positionExtrema := output.trajectory.profiles[2].positionExtrema();
AssertEquals_LREAL(0.22338925049474447904, positionExtrema.Tmax, 1E-9, message:='Profile[2] Tmax incorrect');
AssertEquals_LREAL(94.47974487226861128875, positionExtrema.Maximum, 1E-9, message:='Profile[2] maximum incorrect');
AssertEquals_LREAL(0.02606362117094545780, positionExtrema.Tmin, 1E-9, message:='Profile[2] Tmin incorrect');
AssertEquals_LREAL(-104.28684661857214166503, positionExtrema.Minimum, 1E-9, message:='Profile[2] minimum incorrect');
   

TEST_FINISHED();
END_METHOD

METHOD Test_Trajectory_32
VAR_INST
  ruckig : Struckig.Ruckig(0.001);
  input : Struckig.InputParameter(3) := (
    Synchronization := SynchronizationType.TimeSync,        
    MaxVelocity := [ 2000.00000000000000000000, 2000.00000000000000000000, 2000.00000000000000000000 ],
    MaxAcceleration := [ 20000.00000000000000000000, 20000.00000000000000000000, 20000.00000000000000000000 ],
    MaxJerk := [ 800000.00000000000000000000, 800000.00000000000000000000, 800000.00000000000000000000 ],
    CurrentPosition := [ -71.32072487430589546875, 75.77874394332496876814, -31.17619673281745917848 ],
    CurrentVelocity := [ -39.37043543026334191381, -314.80982911633589083067, -743.63983854388607142027 ],
    CurrentAcceleration := [ 918.61171848468075040728, -8240.24070744882010330912, 376.40421615367449703626 ],
    TargetPosition := [ -38.32577323859909057546, 76.88839801585137934126, 77.24450399202348194194 ],
    TargetVelocity := [ 0.00000000000000000000, 0.00000000000000000000, 0.00000000000000000000 ],
    TargetAcceleration := [ 0.00000000000000000000, 0.00000000000000000000, 0.00000000000000000000 ]
  );
  output : Struckig.OutputParameter;
  positionExtrema : Struckig.PositionExtremaDesc;
END_VAR
TEST('Trajectory_32');

ruckig.update(input, output);

// Check total duration of profiles
AssertEquals_LREAL(Expected := 0.22561874467077386308, Actual := output.Trajectory.Duration, DELTA := 1E-8, Message := 'Duration incorrect');

// Check duration for each phase
positionExtrema := output.trajectory.profiles[0].positionExtrema();
AssertEquals_LREAL(0.22561874467077389084, positionExtrema.Tmax, 1E-9, message:='Profile[0] Tmax incorrect');
AssertEquals_LREAL(-38.32577323859909057546, positionExtrema.Maximum, 1E-9, message:='Profile[0] maximum incorrect');
AssertEquals_LREAL(0.00883895720172546244, positionExtrema.Tmin, 1E-9, message:='Profile[0] Tmin incorrect');
AssertEquals_LREAL(-71.54075918203305661791, positionExtrema.Minimum, 1E-9, message:='Profile[0] minimum incorrect');

positionExtrema := output.trajectory.profiles[1].positionExtrema();
AssertEquals_LREAL(0.22561874448389260261, positionExtrema.Tmax, 1E-9, message:='Profile[1] Tmax incorrect');
AssertEquals_LREAL(76.88839801585137934126, positionExtrema.Maximum, 1E-9, message:='Profile[1] maximum incorrect');
AssertEquals_LREAL(0.04326693976782886031, positionExtrema.Tmin, 1E-9, message:='Profile[1] Tmin incorrect');
AssertEquals_LREAL(64.99037106700389188063, positionExtrema.Minimum, 1E-9, message:='Profile[1] minimum incorrect');

positionExtrema := output.trajectory.profiles[2].positionExtrema();
AssertEquals_LREAL(0.22561874467077386308, positionExtrema.Tmax, 1E-9, message:='Profile[2] Tmax incorrect');
AssertEquals_LREAL(77.24450399202348194194, positionExtrema.Maximum, 1E-9, message:='Profile[2] maximum incorrect');
AssertEquals_LREAL(0.02452949472980790746, positionExtrema.Tmin, 1E-9, message:='Profile[2] Tmin incorrect');
AssertEquals_LREAL(-47.33615887649365561174, positionExtrema.Minimum, 1E-9, message:='Profile[2] minimum incorrect');
   

TEST_FINISHED();
END_METHOD

METHOD Test_Trajectory_33
VAR_INST
  ruckig : Struckig.Ruckig(0.001);
  input : Struckig.InputParameter(3) := (
    Synchronization := SynchronizationType.TimeSync,        
    MaxVelocity := [ 2000.00000000000000000000, 2000.00000000000000000000, 2000.00000000000000000000 ],
    MaxAcceleration := [ 20000.00000000000000000000, 20000.00000000000000000000, 20000.00000000000000000000 ],
    MaxJerk := [ 800000.00000000000000000000, 800000.00000000000000000000, 800000.00000000000000000000 ],
    CurrentPosition := [ -10.72081173000827902797, -58.44147038088563306246, 98.86324493851924444243 ],
    CurrentVelocity := [ -408.47451658779903027607, -786.19958599415508615493, -998.10812621012325962511 ],
    CurrentAcceleration := [ 3503.92425371204808470793, 3035.68280271572984929662, -8529.36175578239635797217 ],
    TargetPosition := [ -24.74505052699171869790, -29.66847304289291287205, -86.07591857423138037575 ],
    TargetVelocity := [ 0.00000000000000000000, 0.00000000000000000000, 0.00000000000000000000 ],
    TargetAcceleration := [ 0.00000000000000000000, 0.00000000000000000000, 0.00000000000000000000 ]
  );
  output : Struckig.OutputParameter;
  positionExtrema : Struckig.PositionExtremaDesc;
END_VAR
TEST('Trajectory_33');

ruckig.update(input, output);

// Check total duration of profiles
AssertEquals_LREAL(Expected := 0.17123630970102474147, Actual := output.Trajectory.Duration, DELTA := 1E-8, Message := 'Duration incorrect');

// Check duration for each phase
positionExtrema := output.trajectory.profiles[0].positionExtrema();
AssertEquals_LREAL(0.00000000000000000000, positionExtrema.Tmax, 1E-9, message:='Profile[0] Tmax incorrect');
AssertEquals_LREAL(-10.72081173000827902797, positionExtrema.Maximum, 1E-9, message:='Profile[0] maximum incorrect');
AssertEquals_LREAL(0.17123630970102476923, positionExtrema.Tmin, 1E-9, message:='Profile[0] Tmin incorrect');
AssertEquals_LREAL(-24.74505052699171869790, positionExtrema.Minimum, 1E-9, message:='Profile[0] minimum incorrect');

positionExtrema := output.trajectory.profiles[1].positionExtrema();
AssertEquals_LREAL(0.17123630970102471371, positionExtrema.Tmax, 1E-9, message:='Profile[1] Tmax incorrect');
AssertEquals_LREAL(-29.66847304289291287205, positionExtrema.Maximum, 1E-9, message:='Profile[1] maximum incorrect');
AssertEquals_LREAL(0.06908515615955748701, positionExtrema.Tmin, 1E-9, message:='Profile[1] Tmin incorrect');
AssertEquals_LREAL(-76.18339289032344652242, positionExtrema.Minimum, 1E-9, message:='Profile[1] minimum incorrect');

positionExtrema := output.trajectory.profiles[2].positionExtrema();
AssertEquals_LREAL(0.00000000000000000000, positionExtrema.Tmax, 1E-9, message:='Profile[2] Tmax incorrect');
AssertEquals_LREAL(98.86324493851924444243, positionExtrema.Maximum, 1E-9, message:='Profile[2] maximum incorrect');
AssertEquals_LREAL(0.17123630970102474147, positionExtrema.Tmin, 1E-9, message:='Profile[2] Tmin incorrect');
AssertEquals_LREAL(-86.07591857423138037575, positionExtrema.Minimum, 1E-9, message:='Profile[2] minimum incorrect');
   

TEST_FINISHED();
END_METHOD

METHOD Test_Trajectory_HasTargetVelocity_34
VAR_INST
  ruckig : Struckig.Ruckig(0.001);
  input : Struckig.InputParameter(3) := (
    Synchronization := SynchronizationType.TimeSync,        
    MaxVelocity := [ 2000.00000000000000000000, 2000.00000000000000000000, 2000.00000000000000000000 ],
    MaxAcceleration := [ 20000.00000000000000000000, 20000.00000000000000000000, 20000.00000000000000000000 ],
    MaxJerk := [ 800000.00000000000000000000, 800000.00000000000000000000, 800000.00000000000000000000 ],
    CurrentPosition := [ 52.72619781679460970736, -25.78201897219773286452, 80.53760009793651875043 ],
    CurrentVelocity := [ -120.69783207836667315860, 178.50171370384009605914, -265.96277737557261389156 ],
    CurrentAcceleration := [ 9869.62339068779328954406, 8236.73224664633380598389, 4587.35631399299018085003 ],
    TargetPosition := [ -7.31302355801524583967, 98.53124939615054245223, -70.22704739896117587250 ],
    TargetVelocity := [ 648.92680228108224582684, 640.55767309494626715605, -28.66025813343185291160 ],
    TargetAcceleration := [ 0.00000000000000000000, 0.00000000000000000000, 0.00000000000000000000 ]
  );
  output : Struckig.OutputParameter;
  positionExtrema : Struckig.PositionExtremaDesc;
END_VAR
TEST('Trajectory_HasTargetVelocity_34');

ruckig.update(input, output);

// Check total duration of profiles
AssertEquals_LREAL(Expected := 0.19340758597333415625, Actual := output.Trajectory.Duration, DELTA := 1E-8, Message := 'Duration incorrect');

// Check duration for each phase
positionExtrema := output.trajectory.profiles[0].positionExtrema();
AssertEquals_LREAL(0.00000000000000000000, positionExtrema.Tmax, 1E-9, message:='Profile[0] Tmax incorrect');
AssertEquals_LREAL(52.72619781679460970736, positionExtrema.Maximum, 1E-9, message:='Profile[0] maximum incorrect');
AssertEquals_LREAL(0.16840758597333416180, positionExtrema.Tmin, 1E-9, message:='Profile[0] Tmin incorrect');
AssertEquals_LREAL(-21.45286028170894354616, positionExtrema.Minimum, 1E-9, message:='Profile[0] minimum incorrect');

positionExtrema := output.trajectory.profiles[1].positionExtrema();
AssertEquals_LREAL(0.19340758597333415625, positionExtrema.Tmax, 1E-9, message:='Profile[1] Tmax incorrect');
AssertEquals_LREAL(98.53124939615054245223, positionExtrema.Maximum, 1E-9, message:='Profile[1] maximum incorrect');
AssertEquals_LREAL(0.00000000000000000000, positionExtrema.Tmin, 1E-9, message:='Profile[1] Tmin incorrect');
AssertEquals_LREAL(-25.78201897219773286452, positionExtrema.Minimum, 1E-9, message:='Profile[1] minimum incorrect');

positionExtrema := output.trajectory.profiles[2].positionExtrema();
AssertEquals_LREAL(0.00000000000000000000, positionExtrema.Tmax, 1E-9, message:='Profile[2] Tmax incorrect');
AssertEquals_LREAL(80.53760009793651875043, positionExtrema.Maximum, 1E-9, message:='Profile[2] maximum incorrect');
AssertEquals_LREAL(0.19340758597333415625, positionExtrema.Tmin, 1E-9, message:='Profile[2] Tmin incorrect');
AssertEquals_LREAL(-70.22704739896117587250, positionExtrema.Minimum, 1E-9, message:='Profile[2] minimum incorrect');
   

TEST_FINISHED();
END_METHOD

METHOD Test_Trajectory_HasTargetVelocity_35
VAR_INST
  ruckig : Struckig.Ruckig(0.001);
  input : Struckig.InputParameter(3) := (
    Synchronization := SynchronizationType.TimeSync,        
    MaxVelocity := [ 2000.00000000000000000000, 2000.00000000000000000000, 2000.00000000000000000000 ],
    MaxAcceleration := [ 20000.00000000000000000000, 20000.00000000000000000000, 20000.00000000000000000000 ],
    MaxJerk := [ 800000.00000000000000000000, 800000.00000000000000000000, 800000.00000000000000000000 ],
    CurrentPosition := [ -34.17551015513085133080, -36.11913195800440234962, 51.20006403327516864010 ],
    CurrentVelocity := [ -436.11356880285654824547, -175.40667275745920505869, 746.11367552095180144534 ],
    CurrentAcceleration := [ -9866.78282408208724518772, -2137.40956356850620068144, 2870.77810427219810662791 ],
    TargetPosition := [ 94.89098874895094581916, -43.87608688101931875281, 99.33475834942979076914 ],
    TargetVelocity := [ 945.80038372223793885496, -169.18944510068342879094, 349.24092684862353053177 ],
    TargetAcceleration := [ 0.00000000000000000000, 0.00000000000000000000, 0.00000000000000000000 ]
  );
  output : Struckig.OutputParameter;
  positionExtrema : Struckig.PositionExtremaDesc;
END_VAR
TEST('Trajectory_HasTargetVelocity_35');

ruckig.update(input, output);

// Check total duration of profiles
AssertEquals_LREAL(Expected := 0.19433376507479860340, Actual := output.Trajectory.Duration, DELTA := 1E-8, Message := 'Duration incorrect');

// Check duration for each phase
positionExtrema := output.trajectory.profiles[0].positionExtrema();
AssertEquals_LREAL(0.19433376507479860340, positionExtrema.Tmax, 1E-9, message:='Profile[0] Tmax incorrect');
AssertEquals_LREAL(94.89098874895094581916, positionExtrema.Maximum, 1E-9, message:='Profile[0] maximum incorrect');
AssertEquals_LREAL(0.03733347853010261091, positionExtrema.Tmin, 1E-9, message:='Profile[0] Tmin incorrect');
AssertEquals_LREAL(-50.39525451816182055609, positionExtrema.Minimum, 1E-9, message:='Profile[0] minimum incorrect');

positionExtrema := output.trajectory.profiles[1].positionExtrema();
AssertEquals_LREAL(0.00000000000000000000, positionExtrema.Tmax, 1E-9, message:='Profile[1] Tmax incorrect');
AssertEquals_LREAL(-36.11913195800440234962, positionExtrema.Maximum, 1E-9, message:='Profile[1] maximum incorrect');
AssertEquals_LREAL(0.19433376507479860340, positionExtrema.Tmin, 1E-9, message:='Profile[1] Tmin incorrect');
AssertEquals_LREAL(-43.87608688101931875281, positionExtrema.Minimum, 1E-9, message:='Profile[1] minimum incorrect');

positionExtrema := output.trajectory.profiles[2].positionExtrema();
AssertEquals_LREAL(0.19433376507479860340, positionExtrema.Tmax, 1E-9, message:='Profile[2] Tmax incorrect');
AssertEquals_LREAL(99.33475834942979076914, positionExtrema.Maximum, 1E-9, message:='Profile[2] maximum incorrect');
AssertEquals_LREAL(0.00000000000000000000, positionExtrema.Tmin, 1E-9, message:='Profile[2] Tmin incorrect');
AssertEquals_LREAL(51.20006403327516864010, positionExtrema.Minimum, 1E-9, message:='Profile[2] minimum incorrect');
   

TEST_FINISHED();
END_METHOD

METHOD Test_Trajectory_HasTargetVelocity_36
VAR_INST
  ruckig : Struckig.Ruckig(0.001);
  input : Struckig.InputParameter(3) := (
    Synchronization := SynchronizationType.TimeSync,        
    MaxVelocity := [ 2000.00000000000000000000, 2000.00000000000000000000, 2000.00000000000000000000 ],
    MaxAcceleration := [ 20000.00000000000000000000, 20000.00000000000000000000, 20000.00000000000000000000 ],
    MaxJerk := [ 800000.00000000000000000000, 800000.00000000000000000000, 800000.00000000000000000000 ],
    CurrentPosition := [ 64.35804589046725254775, -17.92542582379405757820, 1.48297994216896711350 ],
    CurrentVelocity := [ 464.92943892208950273925, -779.25597761349285974575, 998.42982599227457285451 ],
    CurrentAcceleration := [ 4749.41918638301285682246, -6355.94416374630964128301, 521.38908747176901670173 ],
    TargetPosition := [ 90.33897695077399703223, -51.53109090258827507114, -18.12118447758692241223 ],
    TargetVelocity := [ 651.93427968717173826008, 22.75188801650608638738, 576.72189974234174769663 ],
    TargetAcceleration := [ 0.00000000000000000000, 0.00000000000000000000, 0.00000000000000000000 ]
  );
  output : Struckig.OutputParameter;
  positionExtrema : Struckig.PositionExtremaDesc;
END_VAR
TEST('Trajectory_HasTargetVelocity_36');

ruckig.update(input, output);

// Check total duration of profiles
AssertEquals_LREAL(Expected := 0.22796271730102146691, Actual := output.Trajectory.Duration, DELTA := 1E-8, Message := 'Duration incorrect');

// Check duration for each phase
positionExtrema := output.trajectory.profiles[0].positionExtrema();
AssertEquals_LREAL(0.22796271730102146691, positionExtrema.Tmax, 1E-9, message:='Profile[0] Tmax incorrect');
AssertEquals_LREAL(90.33897695077399703223, positionExtrema.Maximum, 1E-9, message:='Profile[0] maximum incorrect');
AssertEquals_LREAL(0.00000000000000000000, positionExtrema.Tmin, 1E-9, message:='Profile[0] Tmin incorrect');
AssertEquals_LREAL(64.35804589046725254775, positionExtrema.Minimum, 1E-9, message:='Profile[0] minimum incorrect');

positionExtrema := output.trajectory.profiles[1].positionExtrema();
AssertEquals_LREAL(0.00000000000000000000, positionExtrema.Tmax, 1E-9, message:='Profile[1] Tmax incorrect');
AssertEquals_LREAL(-17.92542582379405757820, positionExtrema.Maximum, 1E-9, message:='Profile[1] maximum incorrect');
AssertEquals_LREAL(0.21997970156554483290, positionExtrema.Tmin, 1E-9, message:='Profile[1] Tmin incorrect');
AssertEquals_LREAL(-51.64657663770686468752, positionExtrema.Minimum, 1E-9, message:='Profile[1] minimum incorrect');

positionExtrema := output.trajectory.profiles[2].positionExtrema();
AssertEquals_LREAL(0.09985417258924977890, positionExtrema.Tmax, 1E-9, message:='Profile[2] Tmax incorrect');
AssertEquals_LREAL(25.50333501341721742506, positionExtrema.Maximum, 1E-9, message:='Profile[2] maximum incorrect');
AssertEquals_LREAL(0.20296271730102147246, positionExtrema.Tmin, 1E-9, message:='Profile[2] Tmin incorrect');
AssertEquals_LREAL(-30.45589863781214745586, positionExtrema.Minimum, 1E-9, message:='Profile[2] minimum incorrect');
   

TEST_FINISHED();
END_METHOD

METHOD Test_Trajectory_HasTargetAcceleration_37
VAR_INST
  ruckig : Struckig.Ruckig(0.001);
  input : Struckig.InputParameter(3) := (
    Synchronization := SynchronizationType.TimeSync,        
    MaxVelocity := [ 2000.00000000000000000000, 2000.00000000000000000000, 2000.00000000000000000000 ],
    MaxAcceleration := [ 20000.00000000000000000000, 20000.00000000000000000000, 20000.00000000000000000000 ],
    MaxJerk := [ 800000.00000000000000000000, 800000.00000000000000000000, 800000.00000000000000000000 ],
    CurrentPosition := [ 75.70258410717627839404, -31.81448222562724481577, -58.08554852109006816363 ],
    CurrentVelocity := [ 171.95882136884461033333, -584.70058950900761374214, 745.12321825604590230796 ],
    CurrentAcceleration := [ 5092.19654988173533638474, 7179.19572851603152230382, 1704.28450887377948674839 ],
    TargetPosition := [ 97.60417669221266123714, 88.97844242319803242935, -19.79432812800784802221 ],
    TargetVelocity := [ 0.00000000000000000000, 0.00000000000000000000, 0.00000000000000000000 ],
    TargetAcceleration := [ 983.95730849860865419032, -389.38723727042054179037, -311.43162034307158592128 ]
  );
  output : Struckig.OutputParameter;
  positionExtrema : Struckig.PositionExtremaDesc;
END_VAR
TEST('Trajectory_HasTargetAcceleration_37');

ruckig.update(input, output);

// Check total duration of profiles
AssertEquals_LREAL(Expected := 0.21113509394885510151, Actual := output.Trajectory.Duration, DELTA := 1E-8, Message := 'Duration incorrect');

// Check duration for each phase
positionExtrema := output.trajectory.profiles[0].positionExtrema();
AssertEquals_LREAL(0.20867520067760855773, positionExtrema.Tmax, 1E-9, message:='Profile[0] Tmax incorrect');
AssertEquals_LREAL(97.60516902544232209493, positionExtrema.Maximum, 1E-9, message:='Profile[0] maximum incorrect');
AssertEquals_LREAL(0.00000000000000000000, positionExtrema.Tmin, 1E-9, message:='Profile[0] Tmin incorrect');
AssertEquals_LREAL(75.70258410717627839404, positionExtrema.Minimum, 1E-9, message:='Profile[0] minimum incorrect');

positionExtrema := output.trajectory.profiles[1].positionExtrema();
AssertEquals_LREAL(0.21113509394885510151, positionExtrema.Tmax, 1E-9, message:='Profile[1] Tmax incorrect');
AssertEquals_LREAL(88.97844242319803242935, positionExtrema.Maximum, 1E-9, message:='Profile[1] maximum incorrect');
AssertEquals_LREAL(0.01602600533935496022, positionExtrema.Tmin, 1E-9, message:='Profile[1] Tmin incorrect');
AssertEquals_LREAL(-39.71416974486287898571, positionExtrema.Minimum, 1E-9, message:='Profile[1] minimum incorrect');

positionExtrema := output.trajectory.profiles[2].positionExtrema();
AssertEquals_LREAL(0.21113509394885504600, positionExtrema.Tmax, 1E-9, message:='Profile[2] Tmax incorrect');
AssertEquals_LREAL(-19.79432812800784091678, positionExtrema.Maximum, 1E-9, message:='Profile[2] maximum incorrect');
AssertEquals_LREAL(0.00000000000000000000, positionExtrema.Tmin, 1E-9, message:='Profile[2] Tmin incorrect');
AssertEquals_LREAL(-58.08554852109006816363, positionExtrema.Minimum, 1E-9, message:='Profile[2] minimum incorrect');
   

TEST_FINISHED();
END_METHOD

METHOD Test_Trajectory_HasTargetVelocity_HasTargetAcceleration_38
VAR_INST
  ruckig : Struckig.Ruckig(0.001);
  input : Struckig.InputParameter(3) := (
    Synchronization := SynchronizationType.TimeSync,        
    MaxVelocity := [ 2000.00000000000000000000, 2000.00000000000000000000, 2000.00000000000000000000 ],
    MaxAcceleration := [ 20000.00000000000000000000, 20000.00000000000000000000, 20000.00000000000000000000 ],
    MaxJerk := [ 800000.00000000000000000000, 800000.00000000000000000000, 800000.00000000000000000000 ],
    CurrentPosition := [ 70.18836201933098095651, -77.67370458831963730972, -11.76145133517785268396 ],
    CurrentVelocity := [ -105.04558581308560860634, 265.56449346599174532457, 964.37814674831179218017 ],
    CurrentAcceleration := [ -6039.95733145092708582524, -2777.20507650207400729414, 4352.81085492715828877408 ],
    TargetPosition := [ 71.40233970199534496714, 5.40303445887771260914, 92.98580498819549688960 ],
    TargetVelocity := [ -236.50355991826609169948, -66.98837676043160627160, 870.41763001953563616553 ],
    TargetAcceleration := [ -500.07275325607560034769, 72.93763981243137095589, -942.49209154303241575690 ]
  );
  output : Struckig.OutputParameter;
  positionExtrema : Struckig.PositionExtremaDesc;
END_VAR
TEST('Trajectory_HasTargetVelocity_HasTargetAcceleration_38');

ruckig.update(input, output);

// Check total duration of profiles
AssertEquals_LREAL(Expected := 0.14901888909886754075, Actual := output.Trajectory.Duration, DELTA := 1E-8, Message := 'Duration incorrect');

// Check duration for each phase
positionExtrema := output.trajectory.profiles[0].positionExtrema();
AssertEquals_LREAL(0.12406814159805865105, positionExtrema.Tmax, 1E-9, message:='Profile[0] Tmax incorrect');
AssertEquals_LREAL(75.12313380408009777511, positionExtrema.Maximum, 1E-9, message:='Profile[0] maximum incorrect');
AssertEquals_LREAL(0.02561480747291104351, positionExtrema.Tmin, 1E-9, message:='Profile[0] Tmin incorrect');
AssertEquals_LREAL(67.75537848504214366585, positionExtrema.Minimum, 1E-9, message:='Profile[0] minimum incorrect');

positionExtrema := output.trajectory.profiles[1].positionExtrema();
AssertEquals_LREAL(0.13598633944686283614, positionExtrema.Tmax, 1E-9, message:='Profile[1] Tmax incorrect');
AssertEquals_LREAL(5.98711873384755755012, positionExtrema.Maximum, 1E-9, message:='Profile[1] maximum incorrect');
AssertEquals_LREAL(0.00000000000000000000, positionExtrema.Tmin, 1E-9, message:='Profile[1] Tmin incorrect');
AssertEquals_LREAL(-77.67370458831963730972, positionExtrema.Minimum, 1E-9, message:='Profile[1] minimum incorrect');

positionExtrema := output.trajectory.profiles[2].positionExtrema();
AssertEquals_LREAL(0.14901888909886754075, positionExtrema.Tmax, 1E-9, message:='Profile[2] Tmax incorrect');
AssertEquals_LREAL(92.98580498819549688960, positionExtrema.Maximum, 1E-9, message:='Profile[2] maximum incorrect');
AssertEquals_LREAL(0.00000000000000000000, positionExtrema.Tmin, 1E-9, message:='Profile[2] Tmin incorrect');
AssertEquals_LREAL(-11.76145133517785268396, positionExtrema.Minimum, 1E-9, message:='Profile[2] minimum incorrect');
   

TEST_FINISHED();
END_METHOD

METHOD Test_Trajectory_HasTargetAcceleration_39
VAR_INST
  ruckig : Struckig.Ruckig(0.001);
  input : Struckig.InputParameter(3) := (
    Synchronization := SynchronizationType.TimeSync,        
    MaxVelocity := [ 2000.00000000000000000000, 2000.00000000000000000000, 2000.00000000000000000000 ],
    MaxAcceleration := [ 20000.00000000000000000000, 20000.00000000000000000000, 20000.00000000000000000000 ],
    MaxJerk := [ 800000.00000000000000000000, 800000.00000000000000000000, 800000.00000000000000000000 ],
    CurrentPosition := [ -21.93974605417949419461, -18.49856402298217972202, -96.65992156980888694306 ],
    CurrentVelocity := [ 560.92968123589912465832, -454.79210991651348194864, -556.36905002756998328550 ],
    CurrentAcceleration := [ 6747.73447463338743546046, 9628.82123479624351602979, 5462.73061834566397010349 ],
    TargetPosition := [ -36.27372063241573840742, 69.45477693939508867516, -56.03831440156044152445 ],
    TargetVelocity := [ 0.00000000000000000000, 0.00000000000000000000, 0.00000000000000000000 ],
    TargetAcceleration := [ 228.31394350642813151353, -518.68886336123591718206, -694.01647177787629061640 ]
  );
  output : Struckig.OutputParameter;
  positionExtrema : Struckig.PositionExtremaDesc;
END_VAR
TEST('Trajectory_HasTargetAcceleration_39');

ruckig.update(input, output);

// Check total duration of profiles
AssertEquals_LREAL(Expected := 0.17804896497402217248, Actual := output.Trajectory.Duration, DELTA := 1E-8, Message := 'Duration incorrect');

// Check duration for each phase
positionExtrema := output.trajectory.profiles[0].positionExtrema();
AssertEquals_LREAL(0.05596801189631349371, positionExtrema.Tmax, 1E-9, message:='Profile[0] Tmax incorrect');
AssertEquals_LREAL(-1.82711489240683677693, positionExtrema.Maximum, 1E-9, message:='Profile[0] maximum incorrect');
AssertEquals_LREAL(0.17804896497402203370, positionExtrema.Tmin, 1E-9, message:='Profile[0] Tmin incorrect');
AssertEquals_LREAL(-36.27372063241574551284, positionExtrema.Minimum, 1E-9, message:='Profile[0] minimum incorrect');

positionExtrema := output.trajectory.profiles[1].positionExtrema();
AssertEquals_LREAL(0.17804896497402217248, positionExtrema.Tmax, 1E-9, message:='Profile[1] Tmax incorrect');
AssertEquals_LREAL(69.45477693939508867516, positionExtrema.Maximum, 1E-9, message:='Profile[1] maximum incorrect');
AssertEquals_LREAL(0.01296397345650469532, positionExtrema.Tmin, 1E-9, message:='Profile[1] Tmin incorrect');
AssertEquals_LREAL(-23.29484015015810172144, positionExtrema.Minimum, 1E-9, message:='Profile[1] minimum incorrect');

positionExtrema := output.trajectory.profiles[2].positionExtrema();
AssertEquals_LREAL(0.17804896497402220024, positionExtrema.Tmax, 1E-9, message:='Profile[2] Tmax incorrect');
AssertEquals_LREAL(-56.03831440156044152445, positionExtrema.Maximum, 1E-9, message:='Profile[2] maximum incorrect');
AssertEquals_LREAL(0.04613976266622405592, positionExtrema.Tmin, 1E-9, message:='Profile[2] Tmin incorrect');
AssertEquals_LREAL(-106.33609120894020350079, positionExtrema.Minimum, 1E-9, message:='Profile[2] minimum incorrect');
   

TEST_FINISHED();
END_METHOD

METHOD Test_Trajectory_40
VAR_INST
  ruckig : Struckig.Ruckig(0.001);
  input : Struckig.InputParameter(3) := (
    Synchronization := SynchronizationType.TimeSync,        
    MaxVelocity := [ 2000.00000000000000000000, 2000.00000000000000000000, 2000.00000000000000000000 ],
    MaxAcceleration := [ 20000.00000000000000000000, 20000.00000000000000000000, 20000.00000000000000000000 ],
    MaxJerk := [ 800000.00000000000000000000, 800000.00000000000000000000, 800000.00000000000000000000 ],
    CurrentPosition := [ 29.38520952151498022431, 0.54024576846694571941, -55.20826603737940274641 ],
    CurrentVelocity := [ -969.77050425776712927473, -274.95655325444397476531, 136.62875181670483470953 ],
    CurrentAcceleration := [ -3024.14261213553436391521, 816.78995976388432609383, -4328.68204209528175852029 ],
    TargetPosition := [ 1.97730433317153142525, -41.44239712071811254646, -63.08579022434781791162 ],
    TargetVelocity := [ 0.00000000000000000000, 0.00000000000000000000, 0.00000000000000000000 ],
    TargetAcceleration := [ 0.00000000000000000000, 0.00000000000000000000, 0.00000000000000000000 ]
  );
  output : Struckig.OutputParameter;
  positionExtrema : Struckig.PositionExtremaDesc;
END_VAR
TEST('Trajectory_40');

ruckig.update(input, output);

// Check total duration of profiles
AssertEquals_LREAL(Expected := 0.13217815288228063064, Actual := output.Trajectory.Duration, DELTA := 1E-8, Message := 'Duration incorrect');

// Check duration for each phase
positionExtrema := output.trajectory.profiles[0].positionExtrema();
AssertEquals_LREAL(0.00000000000000000000, positionExtrema.Tmax, 1E-9, message:='Profile[0] Tmax incorrect');
AssertEquals_LREAL(29.38520952151498022431, positionExtrema.Maximum, 1E-9, message:='Profile[0] maximum incorrect');
AssertEquals_LREAL(0.06794606535212494025, positionExtrema.Tmin, 1E-9, message:='Profile[0] Tmin incorrect');
AssertEquals_LREAL(-9.67357879957821609196, positionExtrema.Minimum, 1E-9, message:='Profile[0] minimum incorrect');

positionExtrema := output.trajectory.profiles[1].positionExtrema();
AssertEquals_LREAL(0.00000000000000000000, positionExtrema.Tmax, 1E-9, message:='Profile[1] Tmax incorrect');
AssertEquals_LREAL(0.54024576846694571941, positionExtrema.Maximum, 1E-9, message:='Profile[1] maximum incorrect');
AssertEquals_LREAL(0.13217815288228063064, positionExtrema.Tmin, 1E-9, message:='Profile[1] Tmin incorrect');
AssertEquals_LREAL(-41.44239712071811254646, positionExtrema.Minimum, 1E-9, message:='Profile[1] minimum incorrect');

positionExtrema := output.trajectory.profiles[2].positionExtrema();
AssertEquals_LREAL(0.01413581147570610458, positionExtrema.Tmax, 1E-9, message:='Profile[2] Tmax incorrect');
AssertEquals_LREAL(-54.08246211603182018735, positionExtrema.Maximum, 1E-9, message:='Profile[2] maximum incorrect');
AssertEquals_LREAL(0.13217815261799065185, positionExtrema.Tmin, 1E-9, message:='Profile[2] Tmin incorrect');
AssertEquals_LREAL(-63.08579022434781791162, positionExtrema.Minimum, 1E-9, message:='Profile[2] minimum incorrect');
   

TEST_FINISHED();
END_METHOD

METHOD Test_Trajectory_HasTargetVelocity_HasTargetAcceleration_41
VAR_INST
  ruckig : Struckig.Ruckig(0.001);
  input : Struckig.InputParameter(3) := (
    Synchronization := SynchronizationType.TimeSync,        
    MaxVelocity := [ 2000.00000000000000000000, 2000.00000000000000000000, 2000.00000000000000000000 ],
    MaxAcceleration := [ 20000.00000000000000000000, 20000.00000000000000000000, 20000.00000000000000000000 ],
    MaxJerk := [ 800000.00000000000000000000, 800000.00000000000000000000, 800000.00000000000000000000 ],
    CurrentPosition := [ 77.70133891525995295524, 7.01592092562633240505, 41.88398938907070601090 ],
    CurrentVelocity := [ -954.47536643469038608600, -572.16261829852851406031, 473.16402135503631143365 ],
    CurrentAcceleration := [ -2847.17654342300011194311, -1889.61698757276462856680, -3110.21768918452016805531 ],
    TargetPosition := [ 92.37579717709354554245, -14.04614057772144519731, -73.88361356505039623244 ],
    TargetVelocity := [ 519.95772801058456025203, 127.89327712966064609645, -380.91422286825297760515 ],
    TargetAcceleration := [ -890.64075852453197512659, 681.51569675393488978443, 390.99828361762297390669 ]
  );
  output : Struckig.OutputParameter;
  positionExtrema : Struckig.PositionExtremaDesc;
END_VAR
TEST('Trajectory_HasTargetVelocity_HasTargetAcceleration_41');

ruckig.update(input, output);

// Check total duration of profiles
AssertEquals_LREAL(Expected := 0.18543052523247699481, Actual := output.Trajectory.Duration, DELTA := 1E-8, Message := 'Duration incorrect');

// Check duration for each phase
positionExtrema := output.trajectory.profiles[0].positionExtrema();
AssertEquals_LREAL(0.18543052523247699481, positionExtrema.Tmax, 1E-9, message:='Profile[0] Tmax incorrect');
AssertEquals_LREAL(92.37579717709354554245, positionExtrema.Maximum, 1E-9, message:='Profile[0] maximum incorrect');
AssertEquals_LREAL(0.07568410654937982041, positionExtrema.Tmin, 1E-9, message:='Profile[0] Tmin incorrect');
AssertEquals_LREAL(41.15768150995504015555, positionExtrema.Minimum, 1E-9, message:='Profile[0] minimum incorrect');

positionExtrema := output.trajectory.profiles[1].positionExtrema();
AssertEquals_LREAL(0.00000000000000000000, positionExtrema.Tmax, 1E-9, message:='Profile[1] Tmax incorrect');
AssertEquals_LREAL(7.01592092562633240505, positionExtrema.Maximum, 1E-9, message:='Profile[1] maximum incorrect');
AssertEquals_LREAL(0.16752625845292970497, positionExtrema.Tmin, 1E-9, message:='Profile[1] Tmin incorrect');
AssertEquals_LREAL(-15.47801998831725711625, positionExtrema.Minimum, 1E-9, message:='Profile[1] minimum incorrect');

positionExtrema := output.trajectory.profiles[2].positionExtrema();
AssertEquals_LREAL(0.02111222788851935261, positionExtrema.Tmax, 1E-9, message:='Profile[2] Tmax incorrect');
AssertEquals_LREAL(49.92568034606993876423, positionExtrema.Maximum, 1E-9, message:='Profile[2] maximum incorrect');
AssertEquals_LREAL(0.18543052523247699481, positionExtrema.Tmin, 1E-9, message:='Profile[2] Tmin incorrect');
AssertEquals_LREAL(-73.88361356505039623244, positionExtrema.Minimum, 1E-9, message:='Profile[2] minimum incorrect');
   

TEST_FINISHED();
END_METHOD

METHOD Test_Trajectory_HasTargetAcceleration_42
VAR_INST
  ruckig : Struckig.Ruckig(0.001);
  input : Struckig.InputParameter(3) := (
    Synchronization := SynchronizationType.TimeSync,        
    MaxVelocity := [ 2000.00000000000000000000, 2000.00000000000000000000, 2000.00000000000000000000 ],
    MaxAcceleration := [ 20000.00000000000000000000, 20000.00000000000000000000, 20000.00000000000000000000 ],
    MaxJerk := [ 800000.00000000000000000000, 800000.00000000000000000000, 800000.00000000000000000000 ],
    CurrentPosition := [ 1.58314797372935345265, 90.58707779544036498010, 7.41484167737418431443 ],
    CurrentVelocity := [ 264.66369378964441239077, -967.86838256043972705811, 875.55912471800957064261 ],
    CurrentAcceleration := [ -5955.60883189429478079546, -8419.85921682317348313518, 8392.40723541911211214028 ],
    TargetPosition := [ -58.56616862494692554719, 73.15314018228875170280, 71.09694589628986705065 ],
    TargetVelocity := [ 0.00000000000000000000, 0.00000000000000000000, 0.00000000000000000000 ],
    TargetAcceleration := [ -714.77249466642297193175, -738.86959085233320365660, -949.40990195438507726067 ]
  );
  output : Struckig.OutputParameter;
  positionExtrema : Struckig.PositionExtremaDesc;
END_VAR
TEST('Trajectory_HasTargetAcceleration_42');

ruckig.update(input, output);

// Check total duration of profiles
AssertEquals_LREAL(Expected := 0.16824213942746521488, Actual := output.Trajectory.Duration, DELTA := 1E-8, Message := 'Duration incorrect');

// Check duration for each phase
positionExtrema := output.trajectory.profiles[0].positionExtrema();
AssertEquals_LREAL(0.01755548896013213109, positionExtrema.Tmax, 1E-9, message:='Profile[0] Tmax incorrect');
AssertEquals_LREAL(4.59030121571332649921, positionExtrema.Maximum, 1E-9, message:='Profile[0] maximum incorrect');
AssertEquals_LREAL(0.16645520819079967501, positionExtrema.Tmin, 1E-9, message:='Profile[0] Tmin incorrect');
AssertEquals_LREAL(-58.56654901772477472832, positionExtrema.Minimum, 1E-9, message:='Profile[0] minimum incorrect');

positionExtrema := output.trajectory.profiles[1].positionExtrema();
AssertEquals_LREAL(0.00000000000000000000, positionExtrema.Tmax, 1E-9, message:='Profile[1] Tmax incorrect');
AssertEquals_LREAL(90.58707779544036498010, positionExtrema.Maximum, 1E-9, message:='Profile[1] maximum incorrect');
AssertEquals_LREAL(0.09014117386002259980, positionExtrema.Tmin, 1E-9, message:='Profile[1] Tmin incorrect');
AssertEquals_LREAL(45.07056608531748764790, positionExtrema.Minimum, 1E-9, message:='Profile[1] minimum incorrect');

positionExtrema := output.trajectory.profiles[2].positionExtrema();
AssertEquals_LREAL(0.13468422806677898818, positionExtrema.Tmax, 1E-9, message:='Profile[2] Tmax incorrect');
AssertEquals_LREAL(73.02284673044322005353, positionExtrema.Maximum, 1E-9, message:='Profile[2] maximum incorrect');
AssertEquals_LREAL(0.00000000000000000000, positionExtrema.Tmin, 1E-9, message:='Profile[2] Tmin incorrect');
AssertEquals_LREAL(7.41484167737418431443, positionExtrema.Minimum, 1E-9, message:='Profile[2] minimum incorrect');
   

TEST_FINISHED();
END_METHOD

METHOD Test_Trajectory_HasTargetAcceleration_43
VAR_INST
  ruckig : Struckig.Ruckig(0.001);
  input : Struckig.InputParameter(3) := (
    Synchronization := SynchronizationType.TimeSync,        
    MaxVelocity := [ 2000.00000000000000000000, 2000.00000000000000000000, 2000.00000000000000000000 ],
    MaxAcceleration := [ 20000.00000000000000000000, 20000.00000000000000000000, 20000.00000000000000000000 ],
    MaxJerk := [ 800000.00000000000000000000, 800000.00000000000000000000, 800000.00000000000000000000 ],
    CurrentPosition := [ 53.13739682938987130001, -22.44298053732963182938, -41.20042774153274223181 ],
    CurrentVelocity := [ -304.98663512538098530058, 35.02037430652057992120, 738.80078152761325327447 ],
    CurrentAcceleration := [ -7270.26712820171451312490, -845.41004591047749272548, -4566.56327336276262940373 ],
    TargetPosition := [ 81.86956314333414752582, 96.25424125499196748024, -65.78248687323761600965 ],
    TargetVelocity := [ 0.00000000000000000000, 0.00000000000000000000, 0.00000000000000000000 ],
    TargetAcceleration := [ -511.94239891635919548207, 447.91143210314089628810, -814.86235086373915237345 ]
  );
  output : Struckig.OutputParameter;
  positionExtrema : Struckig.PositionExtremaDesc;
END_VAR
TEST('Trajectory_HasTargetAcceleration_43');

ruckig.update(input, output);

// Check total duration of profiles
AssertEquals_LREAL(Expected := 0.18070492746146707419, Actual := output.Trajectory.Duration, DELTA := 1E-8, Message := 'Duration incorrect');

// Check duration for each phase
positionExtrema := output.trajectory.profiles[0].positionExtrema();
AssertEquals_LREAL(0.18070492746146707419, positionExtrema.Tmax, 1E-9, message:='Profile[0] Tmax incorrect');
AssertEquals_LREAL(81.86956314333414752582, positionExtrema.Maximum, 1E-9, message:='Profile[0] maximum incorrect');
AssertEquals_LREAL(0.03408783391025214243, positionExtrema.Tmin, 1E-9, message:='Profile[0] Tmin incorrect');
AssertEquals_LREAL(43.79836178330638318812, positionExtrema.Minimum, 1E-9, message:='Profile[0] minimum incorrect');

positionExtrema := output.trajectory.profiles[1].positionExtrema();
AssertEquals_LREAL(0.17958514888120891140, positionExtrema.Tmax, 1E-9, message:='Profile[1] Tmax incorrect');
AssertEquals_LREAL(96.25433486131980487244, positionExtrema.Maximum, 1E-9, message:='Profile[1] maximum incorrect');
AssertEquals_LREAL(0.00000000000000000000, positionExtrema.Tmin, 1E-9, message:='Profile[1] Tmin incorrect');
AssertEquals_LREAL(-22.44298053732963182938, positionExtrema.Minimum, 1E-9, message:='Profile[1] minimum incorrect');

positionExtrema := output.trajectory.profiles[2].positionExtrema();
AssertEquals_LREAL(0.05355512909515708353, positionExtrema.Tmax, 1E-9, message:='Profile[2] Tmax incorrect');
AssertEquals_LREAL(-23.29997654589049815854, positionExtrema.Maximum, 1E-9, message:='Profile[2] maximum incorrect');
AssertEquals_LREAL(0.17866777158430743877, positionExtrema.Tmin, 1E-9, message:='Profile[2] Tmin incorrect');
AssertEquals_LREAL(-65.78305048691605350086, positionExtrema.Minimum, 1E-9, message:='Profile[2] minimum incorrect');
   

TEST_FINISHED();
END_METHOD

METHOD Test_Trajectory_HasTargetVelocity_44
VAR_INST
  ruckig : Struckig.Ruckig(0.001);
  input : Struckig.InputParameter(3) := (
    Synchronization := SynchronizationType.TimeSync,        
    MaxVelocity := [ 2000.00000000000000000000, 2000.00000000000000000000, 2000.00000000000000000000 ],
    MaxAcceleration := [ 20000.00000000000000000000, 20000.00000000000000000000, 20000.00000000000000000000 ],
    MaxJerk := [ 800000.00000000000000000000, 800000.00000000000000000000, 800000.00000000000000000000 ],
    CurrentPosition := [ 33.20927605983496277986, 90.97207853642058239529, -55.08094735406923092569 ],
    CurrentVelocity := [ -992.30424733188726804656, -901.32445813848187299300, 586.66877088523051497759 ],
    CurrentAcceleration := [ -2055.28947681546742387582, -6947.94625488244855660014, 5257.19066749439298291691 ],
    TargetPosition := [ 67.40661968603291143154, 85.00720295179675645159, 88.22002633481628208756 ],
    TargetVelocity := [ -402.53524157043091236119, -775.84245093694903516734, -256.32808117758236221562 ],
    TargetAcceleration := [ 0.00000000000000000000, 0.00000000000000000000, 0.00000000000000000000 ]
  );
  output : Struckig.OutputParameter;
  positionExtrema : Struckig.PositionExtremaDesc;
END_VAR
TEST('Trajectory_HasTargetVelocity_44');

ruckig.update(input, output);

// Check total duration of profiles
AssertEquals_LREAL(Expected := 0.23151950260302325835, Actual := output.Trajectory.Duration, DELTA := 1E-8, Message := 'Duration incorrect');

// Check duration for each phase
positionExtrema := output.trajectory.profiles[0].positionExtrema();
AssertEquals_LREAL(0.20651950260302323614, positionExtrema.Tmax, 1E-9, message:='Profile[0] Tmax incorrect');
AssertEquals_LREAL(75.38666739196018795610, positionExtrema.Maximum, 1E-9, message:='Profile[0] maximum incorrect');
AssertEquals_LREAL(0.10082888716067818502, positionExtrema.Tmin, 1E-9, message:='Profile[0] Tmin incorrect');
AssertEquals_LREAL(6.96062616300369274569, positionExtrema.Minimum, 1E-9, message:='Profile[0] minimum incorrect');

positionExtrema := output.trajectory.profiles[1].positionExtrema();
AssertEquals_LREAL(0.20651950260302326390, positionExtrema.Tmax, 1E-9, message:='Profile[1] Tmax incorrect');
AssertEquals_LREAL(102.31993089188715373439, positionExtrema.Maximum, 1E-9, message:='Profile[1] maximum incorrect');
AssertEquals_LREAL(0.09899354847148797432, positionExtrema.Tmin, 1E-9, message:='Profile[1] Tmin incorrect');
AssertEquals_LREAL(59.91000069944395534094, positionExtrema.Minimum, 1E-9, message:='Profile[1] minimum incorrect');

positionExtrema := output.trajectory.profiles[2].positionExtrema();
AssertEquals_LREAL(0.20651950260302326390, positionExtrema.Tmax, 1E-9, message:='Profile[2] Tmax incorrect');
AssertEquals_LREAL(92.54489503092254665262, positionExtrema.Maximum, 1E-9, message:='Profile[2] maximum incorrect');
AssertEquals_LREAL(0.00000000000000000000, positionExtrema.Tmin, 1E-9, message:='Profile[2] Tmin incorrect');
AssertEquals_LREAL(-55.08094735406923092569, positionExtrema.Minimum, 1E-9, message:='Profile[2] minimum incorrect');
   

TEST_FINISHED();
END_METHOD

METHOD Test_Trajectory_HasTargetVelocity_45
VAR_INST
  ruckig : Struckig.Ruckig(0.001);
  input : Struckig.InputParameter(3) := (
    Synchronization := SynchronizationType.TimeSync,        
    MaxVelocity := [ 2000.00000000000000000000, 2000.00000000000000000000, 2000.00000000000000000000 ],
    MaxAcceleration := [ 20000.00000000000000000000, 20000.00000000000000000000, 20000.00000000000000000000 ],
    MaxJerk := [ 800000.00000000000000000000, 800000.00000000000000000000, 800000.00000000000000000000 ],
    CurrentPosition := [ 94.90826698124541849211, 98.68601680143464704997, -94.06931326171563512162 ],
    CurrentVelocity := [ -430.89473663668559311191, -312.79662986488631304383, -992.83444762482452006225 ],
    CurrentAcceleration := [ -5676.65368720607239083620, -3762.56637347724063147325, 6550.62068049420850002207 ],
    TargetPosition := [ -39.76061431821072034154, -54.28480859989317508507, 99.44666750072161676144 ],
    TargetVelocity := [ -859.34940974039534467011, 795.33260348280805374088, -780.22698676244044690975 ],
    TargetAcceleration := [ 0.00000000000000000000, 0.00000000000000000000, 0.00000000000000000000 ]
  );
  output : Struckig.OutputParameter;
  positionExtrema : Struckig.PositionExtremaDesc;
END_VAR
TEST('Trajectory_HasTargetVelocity_45');

ruckig.update(input, output);

// Check total duration of profiles
AssertEquals_LREAL(Expected := 0.33133845625565350179, Actual := output.Trajectory.Duration, DELTA := 1E-8, Message := 'Duration incorrect');

// Check duration for each phase
positionExtrema := output.trajectory.profiles[0].positionExtrema();
AssertEquals_LREAL(0.00000000000000000000, positionExtrema.Tmax, 1E-9, message:='Profile[0] Tmax incorrect');
AssertEquals_LREAL(94.90826698124541849211, positionExtrema.Maximum, 1E-9, message:='Profile[0] maximum incorrect');
AssertEquals_LREAL(0.33133845625565355730, positionExtrema.Tmin, 1E-9, message:='Profile[0] Tmin incorrect');
AssertEquals_LREAL(-39.76061431821072034154, positionExtrema.Minimum, 1E-9, message:='Profile[0] minimum incorrect');

positionExtrema := output.trajectory.profiles[1].positionExtrema();
AssertEquals_LREAL(0.00000000000000000000, positionExtrema.Tmax, 1E-9, message:='Profile[1] Tmax incorrect');
AssertEquals_LREAL(98.68601680143464704997, positionExtrema.Maximum, 1E-9, message:='Profile[1] maximum incorrect');
AssertEquals_LREAL(0.25596921475835221482, positionExtrema.Tmin, 1E-9, message:='Profile[1] Tmin incorrect');
AssertEquals_LREAL(-74.18217506467304644957, positionExtrema.Minimum, 1E-9, message:='Profile[1] minimum incorrect');

positionExtrema := output.trajectory.profiles[2].positionExtrema();
AssertEquals_LREAL(0.30633845625565347959, positionExtrema.Tmax, 1E-9, message:='Profile[2] Tmax incorrect');
AssertEquals_LREAL(116.86900883644932491734, positionExtrema.Maximum, 1E-9, message:='Profile[2] maximum incorrect');
AssertEquals_LREAL(0.01681172414938223933, positionExtrema.Tmin, 1E-9, message:='Profile[2] Tmin incorrect');
AssertEquals_LREAL(-109.20131569941064242357, positionExtrema.Minimum, 1E-9, message:='Profile[2] minimum incorrect');
   

TEST_FINISHED();
END_METHOD

METHOD Test_Trajectory_HasTargetVelocity_HasTargetAcceleration_46
VAR_INST
  ruckig : Struckig.Ruckig(0.001);
  input : Struckig.InputParameter(3) := (
    Synchronization := SynchronizationType.TimeSync,        
    MaxVelocity := [ 2000.00000000000000000000, 2000.00000000000000000000, 2000.00000000000000000000 ],
    MaxAcceleration := [ 20000.00000000000000000000, 20000.00000000000000000000, 20000.00000000000000000000 ],
    MaxJerk := [ 800000.00000000000000000000, 800000.00000000000000000000, 800000.00000000000000000000 ],
    CurrentPosition := [ -81.70058267564624543411, -19.21897702137916041920, 94.53377990477645198553 ],
    CurrentVelocity := [ 791.96608977333426082623, 567.98007664216197554197, 949.19373974938935134560 ],
    CurrentAcceleration := [ -9852.41254141048739256803, -751.99368634466736693867, 3617.41551680202064744662 ],
    TargetPosition := [ 4.61526430014728816786, 47.19472748930556349478, -27.25527375543330776964 ],
    TargetVelocity := [ -365.39593288733976805815, -832.73312185042618693842, 15.48785727174674775597 ],
    TargetAcceleration := [ 393.54024330782590368472, -760.25458815149545444001, 23.06111995903222577908 ]
  );
  output : Struckig.OutputParameter;
  positionExtrema : Struckig.PositionExtremaDesc;
END_VAR
TEST('Trajectory_HasTargetVelocity_HasTargetAcceleration_46');

ruckig.update(input, output);

// Check total duration of profiles
AssertEquals_LREAL(Expected := 0.25941536116832880632, Actual := output.Trajectory.Duration, DELTA := 1E-8, Message := 'Duration incorrect');

// Check duration for each phase
positionExtrema := output.trajectory.profiles[0].positionExtrema();
AssertEquals_LREAL(0.23392343586419403478, positionExtrema.Tmax, 1E-9, message:='Profile[0] Tmax incorrect');
AssertEquals_LREAL(11.84902844379517183881, positionExtrema.Maximum, 1E-9, message:='Profile[0] maximum incorrect');
AssertEquals_LREAL(0.00000000000000000000, positionExtrema.Tmin, 1E-9, message:='Profile[0] Tmin incorrect');
AssertEquals_LREAL(-81.70058267564624543411, positionExtrema.Minimum, 1E-9, message:='Profile[0] minimum incorrect');

positionExtrema := output.trajectory.profiles[1].positionExtrema();
AssertEquals_LREAL(0.19491405447314413824, positionExtrema.Tmax, 1E-9, message:='Profile[1] Tmax incorrect');
AssertEquals_LREAL(72.37093782213797510394, positionExtrema.Maximum, 1E-9, message:='Profile[1] maximum incorrect');
AssertEquals_LREAL(0.00000000000000000000, positionExtrema.Tmin, 1E-9, message:='Profile[1] Tmin incorrect');
AssertEquals_LREAL(-19.21897702137916041920, positionExtrema.Minimum, 1E-9, message:='Profile[1] minimum incorrect');

positionExtrema := output.trajectory.profiles[2].positionExtrema();
AssertEquals_LREAL(0.02952176939600252917, positionExtrema.Tmax, 1E-9, message:='Profile[2] Tmax incorrect');
AssertEquals_LREAL(120.70144362619019773319, positionExtrema.Maximum, 1E-9, message:='Profile[2] maximum incorrect');
AssertEquals_LREAL(0.25322160979530433655, positionExtrema.Tmin, 1E-9, message:='Profile[2] Tmin incorrect');
AssertEquals_LREAL(-27.31907826634350300310, positionExtrema.Minimum, 1E-9, message:='Profile[2] minimum incorrect');
   

TEST_FINISHED();
END_METHOD

METHOD Test_Trajectory_HasTargetVelocity_HasTargetAcceleration_47
VAR_INST
  ruckig : Struckig.Ruckig(0.001);
  input : Struckig.InputParameter(3) := (
    Synchronization := SynchronizationType.TimeSync,        
    MaxVelocity := [ 2000.00000000000000000000, 2000.00000000000000000000, 2000.00000000000000000000 ],
    MaxAcceleration := [ 20000.00000000000000000000, 20000.00000000000000000000, 20000.00000000000000000000 ],
    MaxJerk := [ 800000.00000000000000000000, 800000.00000000000000000000, 800000.00000000000000000000 ],
    CurrentPosition := [ 81.61368863479273727535, 18.81647567172932156154, -89.15971183512543518646 ],
    CurrentVelocity := [ 614.05723536338791745948, 343.05287387529847364931, -371.00163086153361291508 ],
    CurrentAcceleration := [ 2762.36060607538092881441, -8252.84383845068077789620, 1522.48694311787949118298 ],
    TargetPosition := [ 31.53792392446635517445, -13.15393306556988761713, -67.81554985684867631335 ],
    TargetVelocity := [ 927.36256285251761255495, -453.39442766394324735302, -734.53754957298599492788 ],
    TargetAcceleration := [ -810.42747656261008160072, 683.82844872197824770410, -296.63416710646515639382 ]
  );
  output : Struckig.OutputParameter;
  positionExtrema : Struckig.PositionExtremaDesc;
END_VAR
TEST('Trajectory_HasTargetVelocity_HasTargetAcceleration_47');

ruckig.update(input, output);

// Check total duration of profiles
AssertEquals_LREAL(Expected := 0.25287606970423076591, Actual := output.Trajectory.Duration, DELTA := 1E-8, Message := 'Duration incorrect');

// Check duration for each phase
positionExtrema := output.trajectory.profiles[0].positionExtrema();
AssertEquals_LREAL(0.02845295075759422462, positionExtrema.Tmax, 1E-9, message:='Profile[0] Tmax incorrect');
AssertEquals_LREAL(97.13230269209392986340, positionExtrema.Maximum, 1E-9, message:='Profile[0] maximum incorrect');
AssertEquals_LREAL(0.22686303535852750390, positionExtrema.Tmin, 1E-9, message:='Profile[0] Tmin incorrect');
AssertEquals_LREAL(9.48720344289291794837, positionExtrema.Minimum, 1E-9, message:='Profile[0] minimum incorrect');

positionExtrema := output.trajectory.profiles[1].positionExtrema();
AssertEquals_LREAL(0.02241468542399701822, positionExtrema.Tmax, 1E-9, message:='Profile[1] Tmax incorrect');
AssertEquals_LREAL(23.03639977720293785524, positionExtrema.Maximum, 1E-9, message:='Profile[1] maximum incorrect');
AssertEquals_LREAL(0.25287606970423076591, positionExtrema.Tmin, 1E-9, message:='Profile[1] Tmin incorrect');
AssertEquals_LREAL(-13.15393306556988761713, positionExtrema.Minimum, 1E-9, message:='Profile[1] minimum incorrect');

positionExtrema := output.trajectory.profiles[2].positionExtrema();
AssertEquals_LREAL(0.20039624088411220337, positionExtrema.Tmax, 1E-9, message:='Profile[2] Tmax incorrect');
AssertEquals_LREAL(-46.06681198459425274905, positionExtrema.Maximum, 1E-9, message:='Profile[2] maximum incorrect');
AssertEquals_LREAL(0.03284040362274634473, positionExtrema.Tmin, 1E-9, message:='Profile[2] Tmin incorrect');
AssertEquals_LREAL(-95.92347928545005686374, positionExtrema.Minimum, 1E-9, message:='Profile[2] minimum incorrect');
   

TEST_FINISHED();
END_METHOD

METHOD Test_Trajectory_HasTargetVelocity_HasTargetAcceleration_48
VAR_INST
  ruckig : Struckig.Ruckig(0.001);
  input : Struckig.InputParameter(3) := (
    Synchronization := SynchronizationType.TimeSync,        
    MaxVelocity := [ 2000.00000000000000000000, 2000.00000000000000000000, 2000.00000000000000000000 ],
    MaxAcceleration := [ 20000.00000000000000000000, 20000.00000000000000000000, 20000.00000000000000000000 ],
    MaxJerk := [ 800000.00000000000000000000, 800000.00000000000000000000, 800000.00000000000000000000 ],
    CurrentPosition := [ -88.66208591478776668282, -31.58880789945652622919, 65.04291982806716987398 ],
    CurrentVelocity := [ 580.03497340359649570019, -746.36896556027750193607, 812.20588456619907447021 ],
    CurrentAcceleration := [ -6519.58462448879436124116, -9252.12079111587627266999, -5505.83185145304014440626 ],
    TargetPosition := [ -85.04127215306982634502, -92.28954144915404356198, -74.37698578032075147348 ],
    TargetVelocity := [ -365.82662455999411577068, -112.69189210154274860543, 154.77689249662125803297 ],
    TargetAcceleration := [ -682.87003825383567345852, -247.18670592987155032461, -122.60845320130738400621 ]
  );
  output : Struckig.OutputParameter;
  positionExtrema : Struckig.PositionExtremaDesc;
END_VAR
TEST('Trajectory_HasTargetVelocity_HasTargetAcceleration_48');

ruckig.update(input, output);

// Check total duration of profiles
AssertEquals_LREAL(Expected := 0.25037129752792702808, Actual := output.Trajectory.Duration, DELTA := 1E-8, Message := 'Duration incorrect');

// Check duration for each phase
positionExtrema := output.trajectory.profiles[0].positionExtrema();
AssertEquals_LREAL(0.04415928948418586242, positionExtrema.Tmax, 1E-9, message:='Profile[0] Tmax incorrect');
AssertEquals_LREAL(-76.79539758143890537667, positionExtrema.Maximum, 1E-9, message:='Profile[0] maximum incorrect');
AssertEquals_LREAL(0.00000000000000000000, positionExtrema.Tmin, 1E-9, message:='Profile[0] Tmin incorrect');
AssertEquals_LREAL(-88.66208591478776668282, positionExtrema.Minimum, 1E-9, message:='Profile[0] minimum incorrect');

positionExtrema := output.trajectory.profiles[1].positionExtrema();
AssertEquals_LREAL(0.00000000000000000000, positionExtrema.Tmax, 1E-9, message:='Profile[1] Tmax incorrect');
AssertEquals_LREAL(-31.58880789945652622919, positionExtrema.Maximum, 1E-9, message:='Profile[1] maximum incorrect');
AssertEquals_LREAL(0.25037129752792697257, positionExtrema.Tmin, 1E-9, message:='Profile[1] Tmin incorrect');
AssertEquals_LREAL(-92.28954144915404356198, positionExtrema.Minimum, 1E-9, message:='Profile[1] minimum incorrect');

positionExtrema := output.trajectory.profiles[2].positionExtrema();
AssertEquals_LREAL(0.01811771018568369973, positionExtrema.Tmax, 1E-9, message:='Profile[2] Tmax incorrect');
AssertEquals_LREAL(78.06162686897538094399, positionExtrema.Maximum, 1E-9, message:='Profile[2] maximum incorrect');
AssertEquals_LREAL(0.23054659268189173216, positionExtrema.Tmin, 1E-9, message:='Profile[2] Tmin incorrect');
AssertEquals_LREAL(-76.43062116116439597135, positionExtrema.Minimum, 1E-9, message:='Profile[2] minimum incorrect');
   

TEST_FINISHED();
END_METHOD

METHOD Test_Trajectory_49
VAR_INST
  ruckig : Struckig.Ruckig(0.001);
  input : Struckig.InputParameter(3) := (
    Synchronization := SynchronizationType.TimeSync,        
    MaxVelocity := [ 2000.00000000000000000000, 2000.00000000000000000000, 2000.00000000000000000000 ],
    MaxAcceleration := [ 20000.00000000000000000000, 20000.00000000000000000000, 20000.00000000000000000000 ],
    MaxJerk := [ 800000.00000000000000000000, 800000.00000000000000000000, 800000.00000000000000000000 ],
    CurrentPosition := [ -29.51211691133248393726, -68.13722912354262462031, 25.86635819923048984492 ],
    CurrentVelocity := [ -361.39127939828188118554, 280.60480492296255761175, 432.98890733596567770292 ],
    CurrentAcceleration := [ -4470.60901176135485002305, 6427.77132791660551447421, -7455.37531375192429550225 ],
    TargetPosition := [ 60.41587137499075765845, -7.73628974565106375394, 93.39422462833789495562 ],
    TargetVelocity := [ 0.00000000000000000000, 0.00000000000000000000, 0.00000000000000000000 ],
    TargetAcceleration := [ 0.00000000000000000000, 0.00000000000000000000, 0.00000000000000000000 ]
  );
  output : Struckig.OutputParameter;
  positionExtrema : Struckig.PositionExtremaDesc;
END_VAR
TEST('Trajectory_49');

ruckig.update(input, output);

// Check total duration of profiles
AssertEquals_LREAL(Expected := 0.19300944274036524462, Actual := output.Trajectory.Duration, DELTA := 1E-8, Message := 'Duration incorrect');

// Check duration for each phase
positionExtrema := output.trajectory.profiles[0].positionExtrema();
AssertEquals_LREAL(0.19300944274036524462, positionExtrema.Tmax, 1E-9, message:='Profile[0] Tmax incorrect');
AssertEquals_LREAL(60.41587137499075765845, positionExtrema.Maximum, 1E-9, message:='Profile[0] maximum incorrect');
AssertEquals_LREAL(0.03058826126470169660, positionExtrema.Tmin, 1E-9, message:='Profile[0] Tmin incorrect');
AssertEquals_LREAL(-38.84193813948969165040, positionExtrema.Minimum, 1E-9, message:='Profile[0] minimum incorrect');

positionExtrema := output.trajectory.profiles[1].positionExtrema();
AssertEquals_LREAL(0.19300944274036524462, positionExtrema.Tmax, 1E-9, message:='Profile[1] Tmax incorrect');
AssertEquals_LREAL(-7.73628974565106375394, positionExtrema.Maximum, 1E-9, message:='Profile[1] maximum incorrect');
AssertEquals_LREAL(0.00000000000000000000, positionExtrema.Tmin, 1E-9, message:='Profile[1] Tmin incorrect');
AssertEquals_LREAL(-68.13722912354262462031, positionExtrema.Minimum, 1E-9, message:='Profile[1] minimum incorrect');

positionExtrema := output.trajectory.profiles[2].positionExtrema();
AssertEquals_LREAL(0.19300944274036524462, positionExtrema.Tmax, 1E-9, message:='Profile[2] Tmax incorrect');
AssertEquals_LREAL(93.39422462833789495562, positionExtrema.Maximum, 1E-9, message:='Profile[2] maximum incorrect');
AssertEquals_LREAL(0.00000000000000000000, positionExtrema.Tmin, 1E-9, message:='Profile[2] Tmin incorrect');
AssertEquals_LREAL(25.86635819923048984492, positionExtrema.Minimum, 1E-9, message:='Profile[2] minimum incorrect');
   

TEST_FINISHED();
END_METHOD

METHOD Test_Trajectory_HasTargetAcceleration_50
VAR_INST
  ruckig : Struckig.Ruckig(0.001);
  input : Struckig.InputParameter(3) := (
    Synchronization := SynchronizationType.TimeSync,        
    MaxVelocity := [ 2000.00000000000000000000, 2000.00000000000000000000, 2000.00000000000000000000 ],
    MaxAcceleration := [ 20000.00000000000000000000, 20000.00000000000000000000, 20000.00000000000000000000 ],
    MaxJerk := [ 800000.00000000000000000000, 800000.00000000000000000000, 800000.00000000000000000000 ],
    CurrentPosition := [ 46.92101107231894729921, -0.50374158461752926996, 29.71857774981103261780 ],
    CurrentVelocity := [ -825.06102637463254723116, 756.18378067008961807005, -198.33013045881875768828 ],
    CurrentAcceleration := [ -4766.41159160333245381480, -5907.94068977043207269162, -2476.07236462418222799897 ],
    TargetPosition := [ 23.42250735434379294020, 12.51307920714354793290, 2.55459165158602274914 ],
    TargetVelocity := [ 0.00000000000000000000, 0.00000000000000000000, 0.00000000000000000000 ],
    TargetAcceleration := [ -489.78938572767407322317, 603.07786572774739397573, -878.19166450623129094311 ]
  );
  output : Struckig.OutputParameter;
  positionExtrema : Struckig.PositionExtremaDesc;
END_VAR
TEST('Trajectory_HasTargetAcceleration_50');

ruckig.update(input, output);

// Check total duration of profiles
AssertEquals_LREAL(Expected := 0.12125503368046111619, Actual := output.Trajectory.Duration, DELTA := 1E-8, Message := 'Duration incorrect');

// Check duration for each phase
positionExtrema := output.trajectory.profiles[0].positionExtrema();
AssertEquals_LREAL(0.00000000000000000000, positionExtrema.Tmax, 1E-9, message:='Profile[0] Tmax incorrect');
AssertEquals_LREAL(46.92101107231894729921, positionExtrema.Maximum, 1E-9, message:='Profile[0] maximum incorrect');
AssertEquals_LREAL(0.06087090854331475565, positionExtrema.Tmin, 1E-9, message:='Profile[0] Tmin incorrect');
AssertEquals_LREAL(14.37204891391303718251, positionExtrema.Minimum, 1E-9, message:='Profile[0] minimum incorrect');

positionExtrema := output.trajectory.profiles[1].positionExtrema();
AssertEquals_LREAL(0.04585205920535920243, positionExtrema.Tmax, 1E-9, message:='Profile[1] Tmax incorrect');
AssertEquals_LREAL(18.22432050158307603738, positionExtrema.Maximum, 1E-9, message:='Profile[1] maximum incorrect');
AssertEquals_LREAL(0.00000000000000000000, positionExtrema.Tmin, 1E-9, message:='Profile[1] Tmin incorrect');
AssertEquals_LREAL(-0.50374158461752926996, positionExtrema.Minimum, 1E-9, message:='Profile[1] minimum incorrect');

positionExtrema := output.trajectory.profiles[2].positionExtrema();
AssertEquals_LREAL(0.00000000000000000000, positionExtrema.Tmax, 1E-9, message:='Profile[2] Tmax incorrect');
AssertEquals_LREAL(29.71857774981103261780, positionExtrema.Maximum, 1E-9, message:='Profile[2] maximum incorrect');
AssertEquals_LREAL(0.11905955451919558730, positionExtrema.Tmin, 1E-9, message:='Profile[2] Tmin incorrect');
AssertEquals_LREAL(2.55388615210469760441, positionExtrema.Minimum, 1E-9, message:='Profile[2] minimum incorrect');
   

TEST_FINISHED();
END_METHOD

METHOD Test_Trajectory_HasTargetVelocity_HasTargetAcceleration_51
VAR_INST
  ruckig : Struckig.Ruckig(0.001);
  input : Struckig.InputParameter(3) := (
    Synchronization := SynchronizationType.TimeSync,        
    MaxVelocity := [ 2000.00000000000000000000, 2000.00000000000000000000, 2000.00000000000000000000 ],
    MaxAcceleration := [ 20000.00000000000000000000, 20000.00000000000000000000, 20000.00000000000000000000 ],
    MaxJerk := [ 800000.00000000000000000000, 800000.00000000000000000000, 800000.00000000000000000000 ],
    CurrentPosition := [ 52.80919631150752024951, -81.68038555889982887948, 42.06917442755320735159 ],
    CurrentVelocity := [ -848.38044536898496517097, -694.53443230755419790512, -67.27027959540748724976 ],
    CurrentAcceleration := [ -7839.42279939661148091545, 2086.65454098016925854608, -1769.91408787331420171540 ],
    TargetPosition := [ 18.36498902426966139956, 7.18108207234031681310, -24.86667965964299753523 ],
    TargetVelocity := [ -484.52530887106502177630, -330.54249305132475456048, 184.78707869201707580942 ],
    TargetAcceleration := [ 34.47472473095945133537, 524.15868234202798703336, 659.72269096659351816925 ]
  );
  output : Struckig.OutputParameter;
  positionExtrema : Struckig.PositionExtremaDesc;
END_VAR
TEST('Trajectory_HasTargetVelocity_HasTargetAcceleration_51');

ruckig.update(input, output);

// Check total duration of profiles
AssertEquals_LREAL(Expected := 0.22814955969060143892, Actual := output.Trajectory.Duration, DELTA := 1E-8, Message := 'Duration incorrect');

// Check duration for each phase
positionExtrema := output.trajectory.profiles[0].positionExtrema();
AssertEquals_LREAL(0.00000000000000000000, positionExtrema.Tmax, 1E-9, message:='Profile[0] Tmax incorrect');
AssertEquals_LREAL(52.80919631150752024951, positionExtrema.Maximum, 1E-9, message:='Profile[0] maximum incorrect');
AssertEquals_LREAL(0.06738171645932469755, positionExtrema.Tmin, 1E-9, message:='Profile[0] Tmin incorrect');
AssertEquals_LREAL(13.99608603958429142722, positionExtrema.Minimum, 1E-9, message:='Profile[0] minimum incorrect');

positionExtrema := output.trajectory.profiles[1].positionExtrema();
AssertEquals_LREAL(0.20249436133767390045, positionExtrema.Tmax, 1E-9, message:='Profile[1] Tmax incorrect');
AssertEquals_LREAL(13.58224981559266097975, positionExtrema.Maximum, 1E-9, message:='Profile[1] maximum incorrect');
AssertEquals_LREAL(0.02239168182377478805, positionExtrema.Tmin, 1E-9, message:='Profile[1] Tmin incorrect');
AssertEquals_LREAL(-95.21214742443424938756, positionExtrema.Minimum, 1E-9, message:='Profile[1] minimum incorrect');

positionExtrema := output.trajectory.profiles[2].positionExtrema();
AssertEquals_LREAL(0.00000000000000000000, positionExtrema.Tmax, 1E-9, message:='Profile[2] Tmax incorrect');
AssertEquals_LREAL(42.06917442755320735159, positionExtrema.Maximum, 1E-9, message:='Profile[2] maximum incorrect');
AssertEquals_LREAL(0.20746496504559683305, positionExtrema.Tmin, 1E-9, message:='Profile[2] Tmin incorrect');
AssertEquals_LREAL(-27.36779954300167716497, positionExtrema.Minimum, 1E-9, message:='Profile[2] minimum incorrect');
   

TEST_FINISHED();
END_METHOD

METHOD Test_Trajectory_HasTargetVelocity_HasTargetAcceleration_52
VAR_INST
  ruckig : Struckig.Ruckig(0.001);
  input : Struckig.InputParameter(3) := (
    Synchronization := SynchronizationType.TimeSync,        
    MaxVelocity := [ 2000.00000000000000000000, 2000.00000000000000000000, 2000.00000000000000000000 ],
    MaxAcceleration := [ 20000.00000000000000000000, 20000.00000000000000000000, 20000.00000000000000000000 ],
    MaxJerk := [ 800000.00000000000000000000, 800000.00000000000000000000, 800000.00000000000000000000 ],
    CurrentPosition := [ 70.08966543358397416341, 67.02576750918015591196, -99.48168571307132879156 ],
    CurrentVelocity := [ 588.65830717227800050750, 212.74254643247036256071, -635.02694193343779716088 ],
    CurrentAcceleration := [ 7993.12948784593754680827, -9408.59304495099058840424, 3250.48874447509660967626 ],
    TargetPosition := [ -7.48002668182049035295, 62.76200784473195426472, -18.86381020756616067047 ],
    TargetVelocity := [ 765.89719739525412478542, -627.93810950196188969130, 726.47320111923500007833 ],
    TargetAcceleration := [ -860.50425738071407977259, 155.49469744486259514815, -721.38398094755166312098 ]
  );
  output : Struckig.OutputParameter;
  positionExtrema : Struckig.PositionExtremaDesc;
END_VAR
TEST('Trajectory_HasTargetVelocity_HasTargetAcceleration_52');

ruckig.update(input, output);

// Check total duration of profiles
AssertEquals_LREAL(Expected := 0.26685118878827923661, Actual := output.Trajectory.Duration, DELTA := 1E-8, Message := 'Duration incorrect');

// Check duration for each phase
positionExtrema := output.trajectory.profiles[0].positionExtrema();
AssertEquals_LREAL(0.03499141185980741975, positionExtrema.Tmax, 1E-9, message:='Profile[0] Tmax incorrect');
AssertEquals_LREAL(89.86858068606741767326, positionExtrema.Maximum, 1E-9, message:='Profile[0] maximum incorrect');
AssertEquals_LREAL(0.24077555846655335214, positionExtrema.Tmin, 1E-9, message:='Profile[0] Tmin incorrect');
AssertEquals_LREAL(-25.37984720034276975298, positionExtrema.Minimum, 1E-9, message:='Profile[0] minimum incorrect');

positionExtrema := output.trajectory.profiles[1].positionExtrema();
AssertEquals_LREAL(0.21928974415401750186, positionExtrema.Tmax, 1E-9, message:='Profile[1] Tmax incorrect');
AssertEquals_LREAL(80.25503967122440940329, positionExtrema.Maximum, 1E-9, message:='Profile[1] maximum incorrect');
AssertEquals_LREAL(0.26685118878827929212, positionExtrema.Tmin, 1E-9, message:='Profile[1] Tmin incorrect');
AssertEquals_LREAL(62.76200784473195426472, positionExtrema.Minimum, 1E-9, message:='Profile[1] minimum incorrect');

positionExtrema := output.trajectory.profiles[2].positionExtrema();
AssertEquals_LREAL(0.26685118878827923661, positionExtrema.Tmax, 1E-9, message:='Profile[2] Tmax incorrect');
AssertEquals_LREAL(-18.86381020756616067047, positionExtrema.Maximum, 1E-9, message:='Profile[2] maximum incorrect');
AssertEquals_LREAL(0.04884648491617400029, positionExtrema.Tmin, 1E-9, message:='Profile[2] Tmin incorrect');
AssertEquals_LREAL(-113.98183572111209116429, positionExtrema.Minimum, 1E-9, message:='Profile[2] minimum incorrect');
   

TEST_FINISHED();
END_METHOD

METHOD Test_Trajectory_53
VAR_INST
  ruckig : Struckig.Ruckig(0.001);
  input : Struckig.InputParameter(3) := (
    Synchronization := SynchronizationType.TimeSync,        
    MaxVelocity := [ 2000.00000000000000000000, 2000.00000000000000000000, 2000.00000000000000000000 ],
    MaxAcceleration := [ 20000.00000000000000000000, 20000.00000000000000000000, 20000.00000000000000000000 ],
    MaxJerk := [ 800000.00000000000000000000, 800000.00000000000000000000, 800000.00000000000000000000 ],
    CurrentPosition := [ 49.63749459770096450484, -62.67069199879444596490, 94.53868838473144364798 ],
    CurrentVelocity := [ 664.16399550988307964872, 189.17863757101872579369, -166.93673264110304899077 ],
    CurrentAcceleration := [ 3813.89534506026757298969, -4230.27473187632494955324, -810.58367009230460098479 ],
    TargetPosition := [ 40.02418382022895571026, 1.64383018244964773658, -62.79757540961892203768 ],
    TargetVelocity := [ 0.00000000000000000000, 0.00000000000000000000, 0.00000000000000000000 ],
    TargetAcceleration := [ 0.00000000000000000000, 0.00000000000000000000, 0.00000000000000000000 ]
  );
  output : Struckig.OutputParameter;
  positionExtrema : Struckig.PositionExtremaDesc;
END_VAR
TEST('Trajectory_53');

ruckig.update(input, output);

// Check total duration of profiles
AssertEquals_LREAL(Expected := 0.19412157092543416703, Actual := output.Trajectory.Duration, DELTA := 1E-8, Message := 'Duration incorrect');

// Check duration for each phase
positionExtrema := output.trajectory.profiles[0].positionExtrema();
AssertEquals_LREAL(0.05226266454630152519, positionExtrema.Tmax, 1E-9, message:='Profile[0] Tmax incorrect');
AssertEquals_LREAL(72.04161381570744993041, positionExtrema.Maximum, 1E-9, message:='Profile[0] maximum incorrect');
AssertEquals_LREAL(0.19412157039685418169, positionExtrema.Tmin, 1E-9, message:='Profile[0] Tmin incorrect');
AssertEquals_LREAL(40.02418382022894860484, positionExtrema.Minimum, 1E-9, message:='Profile[0] minimum incorrect');

positionExtrema := output.trajectory.profiles[1].positionExtrema();
AssertEquals_LREAL(0.19412157092543416703, positionExtrema.Tmax, 1E-9, message:='Profile[1] Tmax incorrect');
AssertEquals_LREAL(1.64383018244964773658, positionExtrema.Maximum, 1E-9, message:='Profile[1] maximum incorrect');
AssertEquals_LREAL(0.00000000000000000000, positionExtrema.Tmin, 1E-9, message:='Profile[1] Tmin incorrect');
AssertEquals_LREAL(-62.67069199879444596490, positionExtrema.Minimum, 1E-9, message:='Profile[1] minimum incorrect');

positionExtrema := output.trajectory.profiles[2].positionExtrema();
AssertEquals_LREAL(0.00000000000000000000, positionExtrema.Tmax, 1E-9, message:='Profile[2] Tmax incorrect');
AssertEquals_LREAL(94.53868838473144364798, positionExtrema.Maximum, 1E-9, message:='Profile[2] maximum incorrect');
AssertEquals_LREAL(0.19412157092543416703, positionExtrema.Tmin, 1E-9, message:='Profile[2] Tmin incorrect');
AssertEquals_LREAL(-62.79757540961892203768, positionExtrema.Minimum, 1E-9, message:='Profile[2] minimum incorrect');
   

TEST_FINISHED();
END_METHOD

METHOD Test_Trajectory_HasTargetVelocity_54
VAR_INST
  ruckig : Struckig.Ruckig(0.001);
  input : Struckig.InputParameter(3) := (
    Synchronization := SynchronizationType.TimeSync,        
    MaxVelocity := [ 2000.00000000000000000000, 2000.00000000000000000000, 2000.00000000000000000000 ],
    MaxAcceleration := [ 20000.00000000000000000000, 20000.00000000000000000000, 20000.00000000000000000000 ],
    MaxJerk := [ 800000.00000000000000000000, 800000.00000000000000000000, 800000.00000000000000000000 ],
    CurrentPosition := [ 97.11911830820099567063, -34.96974423375549179127, -12.00449667266771314189 ],
    CurrentVelocity := [ 732.45673588056706648786, -364.10592093846560146631, 417.20885103824889483803 ],
    CurrentAcceleration := [ -7499.05473487195013149176, -3391.82282403053886810085, -1045.80444633833030820824 ],
    TargetPosition := [ -34.58240005713176401514, -14.14677543732022968470, -36.27520430827089370496 ],
    TargetVelocity := [ -912.82558763807946888846, 208.36586640296604855394, -568.50539307151495904691 ],
    TargetAcceleration := [ 0.00000000000000000000, 0.00000000000000000000, 0.00000000000000000000 ]
  );
  output : Struckig.OutputParameter;
  positionExtrema : Struckig.PositionExtremaDesc;
END_VAR
TEST('Trajectory_HasTargetVelocity_54');

ruckig.update(input, output);

// Check total duration of profiles
AssertEquals_LREAL(Expected := 0.18808008069304424370, Actual := output.Trajectory.Duration, DELTA := 1E-8, Message := 'Duration incorrect');

// Check duration for each phase
positionExtrema := output.trajectory.profiles[0].positionExtrema();
AssertEquals_LREAL(0.01562618158141006186, positionExtrema.Tmax, 1E-9, message:='Profile[0] Tmax incorrect');
AssertEquals_LREAL(107.14032815468360126943, positionExtrema.Maximum, 1E-9, message:='Profile[0] maximum incorrect');
AssertEquals_LREAL(0.18808008069304424370, positionExtrema.Tmin, 1E-9, message:='Profile[0] Tmin incorrect');
AssertEquals_LREAL(-34.58240005713176401514, positionExtrema.Minimum, 1E-9, message:='Profile[0] minimum incorrect');

positionExtrema := output.trajectory.profiles[1].positionExtrema();
AssertEquals_LREAL(0.18808008069304424370, positionExtrema.Tmax, 1E-9, message:='Profile[1] Tmax incorrect');
AssertEquals_LREAL(-14.14677543732022968470, positionExtrema.Maximum, 1E-9, message:='Profile[1] maximum incorrect');
AssertEquals_LREAL(0.03540881837579783198, positionExtrema.Tmin, 1E-9, message:='Profile[1] Tmin incorrect');
AssertEquals_LREAL(-44.10216499913330778782, positionExtrema.Minimum, 1E-9, message:='Profile[1] minimum incorrect');

positionExtrema := output.trajectory.profiles[2].positionExtrema();
AssertEquals_LREAL(0.03261360243271873433, positionExtrema.Tmax, 1E-9, message:='Profile[2] Tmax incorrect');
AssertEquals_LREAL(-3.46659095127397254288, positionExtrema.Maximum, 1E-9, message:='Profile[2] maximum incorrect');
AssertEquals_LREAL(0.18808008069304424370, positionExtrema.Tmin, 1E-9, message:='Profile[2] Tmin incorrect');
AssertEquals_LREAL(-36.27520430827089370496, positionExtrema.Minimum, 1E-9, message:='Profile[2] minimum incorrect');
   

TEST_FINISHED();
END_METHOD

METHOD Test_Trajectory_HasTargetVelocity_55
VAR_INST
  ruckig : Struckig.Ruckig(0.001);
  input : Struckig.InputParameter(3) := (
    Synchronization := SynchronizationType.TimeSync,        
    MaxVelocity := [ 2000.00000000000000000000, 2000.00000000000000000000, 2000.00000000000000000000 ],
    MaxAcceleration := [ 20000.00000000000000000000, 20000.00000000000000000000, 20000.00000000000000000000 ],
    MaxJerk := [ 800000.00000000000000000000, 800000.00000000000000000000, 800000.00000000000000000000 ],
    CurrentPosition := [ 93.14320777040134657909, -89.74312540741888710727, -99.44513086937998025405 ],
    CurrentVelocity := [ 358.10280009786106347747, 608.03888639331830745505, 352.36242097628496594552 ],
    CurrentAcceleration := [ 2330.07739343047796864994, 9276.80286875897945719771, 5318.79396039618404756766 ],
    TargetPosition := [ 90.69471017690091230179, -41.60077247517397580623, 88.58596356723177223103 ],
    TargetVelocity := [ -791.02326773343907007074, -519.34342102358630199888, -658.93165900614667407353 ],
    TargetAcceleration := [ 0.00000000000000000000, 0.00000000000000000000, 0.00000000000000000000 ]
  );
  output : Struckig.OutputParameter;
  positionExtrema : Struckig.PositionExtremaDesc;
END_VAR
TEST('Trajectory_HasTargetVelocity_55');

ruckig.update(input, output);

// Check total duration of profiles
AssertEquals_LREAL(Expected := 0.24005299536906613000, Actual := output.Trajectory.Duration, DELTA := 1E-8, Message := 'Duration incorrect');

// Check duration for each phase
positionExtrema := output.trajectory.profiles[0].positionExtrema();
AssertEquals_LREAL(0.18612405983992955094, positionExtrema.Tmax, 1E-9, message:='Profile[0] Tmax incorrect');
AssertEquals_LREAL(115.79065190073221458533, positionExtrema.Maximum, 1E-9, message:='Profile[0] maximum incorrect');
AssertEquals_LREAL(0.24005299536906613000, positionExtrema.Tmin, 1E-9, message:='Profile[0] Tmin incorrect');
AssertEquals_LREAL(90.69471017690091230179, positionExtrema.Minimum, 1E-9, message:='Profile[0] minimum incorrect');

positionExtrema := output.trajectory.profiles[1].positionExtrema();
AssertEquals_LREAL(0.20158118915996722786, positionExtrema.Tmax, 1E-9, message:='Profile[1] Tmax incorrect');
AssertEquals_LREAL(-28.88685866039741512168, positionExtrema.Maximum, 1E-9, message:='Profile[1] maximum incorrect');
AssertEquals_LREAL(0.00000000000000000000, positionExtrema.Tmin, 1E-9, message:='Profile[1] Tmin incorrect');
AssertEquals_LREAL(-89.74312540741888710727, positionExtrema.Minimum, 1E-9, message:='Profile[1] minimum incorrect');

positionExtrema := output.trajectory.profiles[2].positionExtrema();
AssertEquals_LREAL(0.21505299536906613556, positionExtrema.Tmax, 1E-9, message:='Profile[2] Tmax incorrect');
AssertEquals_LREAL(102.97592170905214459253, positionExtrema.Maximum, 1E-9, message:='Profile[2] maximum incorrect');
AssertEquals_LREAL(0.00000000000000000000, positionExtrema.Tmin, 1E-9, message:='Profile[2] Tmin incorrect');
AssertEquals_LREAL(-99.44513086937998025405, positionExtrema.Minimum, 1E-9, message:='Profile[2] minimum incorrect');
   

TEST_FINISHED();
END_METHOD

METHOD Test_Trajectory_HasTargetVelocity_HasTargetAcceleration_56
VAR_INST
  ruckig : Struckig.Ruckig(0.001);
  input : Struckig.InputParameter(3) := (
    Synchronization := SynchronizationType.TimeSync,        
    MaxVelocity := [ 2000.00000000000000000000, 2000.00000000000000000000, 2000.00000000000000000000 ],
    MaxAcceleration := [ 20000.00000000000000000000, 20000.00000000000000000000, 20000.00000000000000000000 ],
    MaxJerk := [ 800000.00000000000000000000, 800000.00000000000000000000, 800000.00000000000000000000 ],
    CurrentPosition := [ -75.10494070961726720270, -6.22395011546019816251, 35.64048680664691914899 ],
    CurrentVelocity := [ -825.41867748520257919154, -559.17669137031361970003, 331.05712850319173412572 ],
    CurrentAcceleration := [ -2748.49249899548522080295, -2734.78689775577458931366, 8828.96129221495357342064 ],
    TargetPosition := [ -88.93249178580995817356, 32.61549251092765189242, -4.33333209618611192582 ],
    TargetVelocity := [ -969.86803709259822880995, 219.52159207481986413768, 145.45315840784223837545 ],
    TargetAcceleration := [ 673.73439439858611876843, 589.54870253816602598818, 268.61037017006333371683 ]
  );
  output : Struckig.OutputParameter;
  positionExtrema : Struckig.PositionExtremaDesc;
END_VAR
TEST('Trajectory_HasTargetVelocity_HasTargetAcceleration_56');

ruckig.update(input, output);

// Check total duration of profiles
AssertEquals_LREAL(Expected := 0.22533279528439006945, Actual := output.Trajectory.Duration, DELTA := 1E-8, Message := 'Duration incorrect');

// Check duration for each phase
positionExtrema := output.trajectory.profiles[0].positionExtrema();
AssertEquals_LREAL(0.13546282954524005437, positionExtrema.Tmax, 1E-9, message:='Profile[0] Tmax incorrect');
AssertEquals_LREAL(-60.83093977470542768060, positionExtrema.Maximum, 1E-9, message:='Profile[0] maximum incorrect');
AssertEquals_LREAL(0.08546282954524006548, positionExtrema.Tmin, 1E-9, message:='Profile[0] Tmin incorrect');
AssertEquals_LREAL(-97.18448406099201974939, positionExtrema.Minimum, 1E-9, message:='Profile[0] minimum incorrect');

positionExtrema := output.trajectory.profiles[1].positionExtrema();
AssertEquals_LREAL(0.22533279528439004169, positionExtrema.Tmax, 1E-9, message:='Profile[1] Tmax incorrect');
AssertEquals_LREAL(32.61549251092765189242, positionExtrema.Maximum, 1E-9, message:='Profile[1] maximum incorrect');
AssertEquals_LREAL(0.04813186201257521613, positionExtrema.Tmin, 1E-9, message:='Profile[1] Tmin incorrect');
AssertEquals_LREAL(-22.45997635018479243740, positionExtrema.Minimum, 1E-9, message:='Profile[1] minimum incorrect');

positionExtrema := output.trajectory.profiles[2].positionExtrema();
AssertEquals_LREAL(0.04893648758049205100, positionExtrema.Tmax, 1E-9, message:='Profile[2] Tmax incorrect');
AssertEquals_LREAL(47.07359821757206930215, positionExtrema.Maximum, 1E-9, message:='Profile[2] maximum incorrect');
AssertEquals_LREAL(0.20659644161609555524, positionExtrema.Tmin, 1E-9, message:='Profile[2] Tmin incorrect');
AssertEquals_LREAL(-6.13445732070238047839, positionExtrema.Minimum, 1E-9, message:='Profile[2] minimum incorrect');
   

TEST_FINISHED();
END_METHOD

METHOD Test_Trajectory_HasTargetAcceleration_57
VAR_INST
  ruckig : Struckig.Ruckig(0.001);
  input : Struckig.InputParameter(3) := (
    Synchronization := SynchronizationType.TimeSync,        
    MaxVelocity := [ 2000.00000000000000000000, 2000.00000000000000000000, 2000.00000000000000000000 ],
    MaxAcceleration := [ 20000.00000000000000000000, 20000.00000000000000000000, 20000.00000000000000000000 ],
    MaxJerk := [ 800000.00000000000000000000, 800000.00000000000000000000, 800000.00000000000000000000 ],
    CurrentPosition := [ -41.78580401739355920654, -54.54341916085618890975, 0.34259842487062996952 ],
    CurrentVelocity := [ 281.70354130105670265038, 551.00897497765049592999, 302.83881748014778167999 ],
    CurrentAcceleration := [ 5924.00492373221095476765, 2065.11081253397605905775, 2773.66158712433571054135 ],
    TargetPosition := [ -35.55043245579965116576, 76.85926955676279703766, -20.12684108733012067205 ],
    TargetVelocity := [ 0.00000000000000000000, 0.00000000000000000000, 0.00000000000000000000 ],
    TargetAcceleration := [ -145.73534974155302279542, -148.36578074146780181763, 565.35337574115942516073 ]
  );
  output : Struckig.OutputParameter;
  positionExtrema : Struckig.PositionExtremaDesc;
END_VAR
TEST('Trajectory_HasTargetAcceleration_57');

ruckig.update(input, output);

// Check total duration of profiles
AssertEquals_LREAL(Expected := 0.16010935183593069664, Actual := output.Trajectory.Duration, DELTA := 1E-8, Message := 'Duration incorrect');

// Check duration for each phase
positionExtrema := output.trajectory.profiles[0].positionExtrema();
AssertEquals_LREAL(0.04108196819819977946, positionExtrema.Tmax, 1E-9, message:='Profile[0] Tmax incorrect');
AssertEquals_LREAL(-33.77372971830767056645, positionExtrema.Maximum, 1E-9, message:='Profile[0] maximum incorrect');
AssertEquals_LREAL(0.00000000000000000000, positionExtrema.Tmin, 1E-9, message:='Profile[0] Tmin incorrect');
AssertEquals_LREAL(-41.78580401739355920654, positionExtrema.Minimum, 1E-9, message:='Profile[0] minimum incorrect');

positionExtrema := output.trajectory.profiles[1].positionExtrema();
AssertEquals_LREAL(0.16010935183593069664, positionExtrema.Tmax, 1E-9, message:='Profile[1] Tmax incorrect');
AssertEquals_LREAL(76.85926955676279703766, positionExtrema.Maximum, 1E-9, message:='Profile[1] maximum incorrect');
AssertEquals_LREAL(0.00000000000000000000, positionExtrema.Tmin, 1E-9, message:='Profile[1] Tmin incorrect');
AssertEquals_LREAL(-54.54341916085618890975, positionExtrema.Minimum, 1E-9, message:='Profile[1] minimum incorrect');

positionExtrema := output.trajectory.profiles[2].positionExtrema();
AssertEquals_LREAL(0.03210937502877184851, positionExtrema.Tmax, 1E-9, message:='Profile[2] Tmax incorrect');
AssertEquals_LREAL(7.08882541134368349134, positionExtrema.Maximum, 1E-9, message:='Profile[2] maximum incorrect');
AssertEquals_LREAL(0.16010935183593069664, positionExtrema.Tmin, 1E-9, message:='Profile[2] Tmin incorrect');
AssertEquals_LREAL(-20.12684108733012067205, positionExtrema.Minimum, 1E-9, message:='Profile[2] minimum incorrect');
   

TEST_FINISHED();
END_METHOD

METHOD Test_Trajectory_HasTargetAcceleration_58
VAR_INST
  ruckig : Struckig.Ruckig(0.001);
  input : Struckig.InputParameter(3) := (
    Synchronization := SynchronizationType.TimeSync,        
    MaxVelocity := [ 2000.00000000000000000000, 2000.00000000000000000000, 2000.00000000000000000000 ],
    MaxAcceleration := [ 20000.00000000000000000000, 20000.00000000000000000000, 20000.00000000000000000000 ],
    MaxJerk := [ 800000.00000000000000000000, 800000.00000000000000000000, 800000.00000000000000000000 ],
    CurrentPosition := [ -28.70185237428661650938, 6.46028600561162136273, 54.49537445608956431897 ],
    CurrentVelocity := [ 444.87185624636094871676, -148.96081495142607309390, -685.59201773629638410057 ],
    CurrentAcceleration := [ -4477.69170784135803842219, -9206.17944268960127374157, -6069.22291510937066050246 ],
    TargetPosition := [ 50.86344209922719983297, 61.53905874524528485381, 55.13748367012033213541 ],
    TargetVelocity := [ 0.00000000000000000000, 0.00000000000000000000, 0.00000000000000000000 ],
    TargetAcceleration := [ -17.25731180548393695062, -728.00753736594913334557, 553.61574831729717516282 ]
  );
  output : Struckig.OutputParameter;
  positionExtrema : Struckig.PositionExtremaDesc;
END_VAR
TEST('Trajectory_HasTargetAcceleration_58');

ruckig.update(input, output);

// Check total duration of profiles
AssertEquals_LREAL(Expected := 0.15873464033901657499, Actual := output.Trajectory.Duration, DELTA := 1E-8, Message := 'Duration incorrect');

// Check duration for each phase
positionExtrema := output.trajectory.profiles[0].positionExtrema();
AssertEquals_LREAL(0.15873464033901651948, positionExtrema.Tmax, 1E-9, message:='Profile[0] Tmax incorrect');
AssertEquals_LREAL(50.86344209922719983297, positionExtrema.Maximum, 1E-9, message:='Profile[0] maximum incorrect');
AssertEquals_LREAL(0.00000000000000000000, positionExtrema.Tmin, 1E-9, message:='Profile[0] Tmin incorrect');
AssertEquals_LREAL(-28.70185237428661650938, positionExtrema.Minimum, 1E-9, message:='Profile[0] minimum incorrect');

positionExtrema := output.trajectory.profiles[1].positionExtrema();
AssertEquals_LREAL(0.15873464033901657499, positionExtrema.Tmax, 1E-9, message:='Profile[1] Tmax incorrect');
AssertEquals_LREAL(61.53905874524528485381, positionExtrema.Maximum, 1E-9, message:='Profile[1] maximum incorrect');
AssertEquals_LREAL(0.03397614115949037367, positionExtrema.Tmin, 1E-9, message:='Profile[1] Tmin incorrect');
AssertEquals_LREAL(1.31497479490398649915, positionExtrema.Minimum, 1E-9, message:='Profile[1] minimum incorrect');

positionExtrema := output.trajectory.profiles[2].positionExtrema();
AssertEquals_LREAL(0.15735060096822323095, positionExtrema.Tmax, 1E-9, message:='Profile[2] Tmax incorrect');
AssertEquals_LREAL(55.13766041794363559347, positionExtrema.Maximum, 1E-9, message:='Profile[2] maximum incorrect');
AssertEquals_LREAL(0.06232337970714629805, positionExtrema.Tmin, 1E-9, message:='Profile[2] Tmin incorrect');
AssertEquals_LREAL(28.75071222396190862014, positionExtrema.Minimum, 1E-9, message:='Profile[2] minimum incorrect');
   

TEST_FINISHED();
END_METHOD

METHOD Test_Trajectory_59
VAR_INST
  ruckig : Struckig.Ruckig(0.001);
  input : Struckig.InputParameter(3) := (
    Synchronization := SynchronizationType.TimeSync,        
    MaxVelocity := [ 2000.00000000000000000000, 2000.00000000000000000000, 2000.00000000000000000000 ],
    MaxAcceleration := [ 20000.00000000000000000000, 20000.00000000000000000000, 20000.00000000000000000000 ],
    MaxJerk := [ 800000.00000000000000000000, 800000.00000000000000000000, 800000.00000000000000000000 ],
    CurrentPosition := [ 48.86656216713086564596, 31.55963588984187140341, -13.09422790776093847853 ],
    CurrentVelocity := [ -274.21841080128081102885, -440.94461360926254656079, -764.75678162210920163488 ],
    CurrentAcceleration := [ -1478.09700836416959646158, 686.79611869591644790489, -9263.72976579731221136171 ],
    TargetPosition := [ 25.57994474955607699940, -15.83091418217283319336, -38.97164514571973370494 ],
    TargetVelocity := [ 0.00000000000000000000, 0.00000000000000000000, 0.00000000000000000000 ],
    TargetAcceleration := [ 0.00000000000000000000, 0.00000000000000000000, 0.00000000000000000000 ]
  );
  output : Struckig.OutputParameter;
  positionExtrema : Struckig.PositionExtremaDesc;
END_VAR
TEST('Trajectory_59');

ruckig.update(input, output);

// Check total duration of profiles
AssertEquals_LREAL(Expected := 0.21566462374557907045, Actual := output.Trajectory.Duration, DELTA := 1E-8, Message := 'Duration incorrect');

// Check duration for each phase
positionExtrema := output.trajectory.profiles[0].positionExtrema();
AssertEquals_LREAL(0.00000000000000000000, positionExtrema.Tmax, 1E-9, message:='Profile[0] Tmax incorrect');
AssertEquals_LREAL(48.86656216713086564596, positionExtrema.Maximum, 1E-9, message:='Profile[0] maximum incorrect');
AssertEquals_LREAL(0.21566462374557909820, positionExtrema.Tmin, 1E-9, message:='Profile[0] Tmin incorrect');
AssertEquals_LREAL(25.57994474955607699940, positionExtrema.Minimum, 1E-9, message:='Profile[0] minimum incorrect');

positionExtrema := output.trajectory.profiles[1].positionExtrema();
AssertEquals_LREAL(0.00000000000000000000, positionExtrema.Tmax, 1E-9, message:='Profile[1] Tmax incorrect');
AssertEquals_LREAL(31.55963588984187140341, positionExtrema.Maximum, 1E-9, message:='Profile[1] maximum incorrect');
AssertEquals_LREAL(0.21566462374557907045, positionExtrema.Tmin, 1E-9, message:='Profile[1] Tmin incorrect');
AssertEquals_LREAL(-15.83091418217285806236, positionExtrema.Minimum, 1E-9, message:='Profile[1] minimum incorrect');

positionExtrema := output.trajectory.profiles[2].positionExtrema();
AssertEquals_LREAL(0.00000000000000000000, positionExtrema.Tmax, 1E-9, message:='Profile[2] Tmax incorrect');
AssertEquals_LREAL(-13.09422790776093847853, positionExtrema.Maximum, 1E-9, message:='Profile[2] maximum incorrect');
AssertEquals_LREAL(0.06757710722237382506, positionExtrema.Tmin, 1E-9, message:='Profile[2] Tmin incorrect');
AssertEquals_LREAL(-48.94577744042891254139, positionExtrema.Minimum, 1E-9, message:='Profile[2] minimum incorrect');
   

TEST_FINISHED();
END_METHOD

METHOD Test_Trajectory_HasTargetVelocity_HasTargetAcceleration_60
VAR_INST
  ruckig : Struckig.Ruckig(0.001);
  input : Struckig.InputParameter(3) := (
    Synchronization := SynchronizationType.TimeSync,        
    MaxVelocity := [ 2000.00000000000000000000, 2000.00000000000000000000, 2000.00000000000000000000 ],
    MaxAcceleration := [ 20000.00000000000000000000, 20000.00000000000000000000, 20000.00000000000000000000 ],
    MaxJerk := [ 800000.00000000000000000000, 800000.00000000000000000000, 800000.00000000000000000000 ],
    CurrentPosition := [ -82.30425131320278353542, 95.77277574475397159404, -0.37873053404373990816 ],
    CurrentVelocity := [ 209.81667767709768668283, 666.24835564548857291811, -156.12978395261052355636 ],
    CurrentAcceleration := [ 554.62083613543836690951, 1781.55274365866716834716, -2304.74829583103382901754 ],
    TargetPosition := [ 78.56604956044506593571, -99.70839917358892989796, -88.26279812419441839211 ],
    TargetVelocity := [ 182.35588906091311400814, 216.59536701599199659540, -100.01197301996137412061 ],
    TargetAcceleration := [ 165.30880475002527418837, -915.29760737648621216067, 984.89234990536533587147 ]
  );
  output : Struckig.OutputParameter;
  positionExtrema : Struckig.PositionExtremaDesc;
END_VAR
TEST('Trajectory_HasTargetVelocity_HasTargetAcceleration_60');

ruckig.update(input, output);

// Check total duration of profiles
AssertEquals_LREAL(Expected := 0.28418047012119368455, Actual := output.Trajectory.Duration, DELTA := 1E-8, Message := 'Duration incorrect');

// Check duration for each phase
positionExtrema := output.trajectory.profiles[0].positionExtrema();
AssertEquals_LREAL(0.28418047012119368455, positionExtrema.Tmax, 1E-9, message:='Profile[0] Tmax incorrect');
AssertEquals_LREAL(78.56604956044506593571, positionExtrema.Maximum, 1E-9, message:='Profile[0] maximum incorrect');
AssertEquals_LREAL(0.00000000000000000000, positionExtrema.Tmin, 1E-9, message:='Profile[0] Tmin incorrect');
AssertEquals_LREAL(-82.30425131320278353542, positionExtrema.Minimum, 1E-9, message:='Profile[0] minimum incorrect');

positionExtrema := output.trajectory.profiles[1].positionExtrema();
AssertEquals_LREAL(0.02722694092957333306, positionExtrema.Tmax, 1E-9, message:='Profile[1] Tmax incorrect');
AssertEquals_LREAL(111.88188475863630344520, positionExtrema.Maximum, 1E-9, message:='Profile[1] maximum incorrect');
AssertEquals_LREAL(0.25973833461914580534, positionExtrema.Tmin, 1E-9, message:='Profile[1] Tmin incorrect');
AssertEquals_LREAL(-103.32890392255741573990, positionExtrema.Minimum, 1E-9, message:='Profile[1] minimum incorrect');

positionExtrema := output.trajectory.profiles[2].positionExtrema();
AssertEquals_LREAL(0.00000000000000000000, positionExtrema.Tmax, 1E-9, message:='Profile[2] Tmax incorrect');
AssertEquals_LREAL(-0.37873053404373990816, positionExtrema.Maximum, 1E-9, message:='Profile[2] maximum incorrect');
AssertEquals_LREAL(0.28418047012119368455, positionExtrema.Tmin, 1E-9, message:='Profile[2] Tmin incorrect');
AssertEquals_LREAL(-88.26279812419441839211, positionExtrema.Minimum, 1E-9, message:='Profile[2] minimum incorrect');
   

TEST_FINISHED();
END_METHOD

METHOD Test_Trajectory_HasTargetVelocity_HasTargetAcceleration_61
VAR_INST
  ruckig : Struckig.Ruckig(0.001);
  input : Struckig.InputParameter(3) := (
    Synchronization := SynchronizationType.TimeSync,        
    MaxVelocity := [ 2000.00000000000000000000, 2000.00000000000000000000, 2000.00000000000000000000 ],
    MaxAcceleration := [ 20000.00000000000000000000, 20000.00000000000000000000, 20000.00000000000000000000 ],
    MaxJerk := [ 800000.00000000000000000000, 800000.00000000000000000000, 800000.00000000000000000000 ],
    CurrentPosition := [ 69.02958196301639759440, -13.39780118806328346182, -96.66107573544628905893 ],
    CurrentVelocity := [ 100.84225227141041614232, -40.44627894454811212199, 363.36834103503497317433 ],
    CurrentAcceleration := [ -7135.55942272971151396632, -622.60760459453013027087, 1671.34292984182866348419 ],
    TargetPosition := [ -16.84074689714994121914, -92.09682308688789476037, -87.06215904519353898650 ],
    TargetVelocity := [ 537.25106843782555188227, -935.18562117857493376505, -396.85249080038204283483 ],
    TargetAcceleration := [ -310.44042758873558796040, -501.02391325450025760802, -57.28028759093501776078 ]
  );
  output : Struckig.OutputParameter;
  positionExtrema : Struckig.PositionExtremaDesc;
END_VAR
TEST('Trajectory_HasTargetVelocity_HasTargetAcceleration_61');

ruckig.update(input, output);

// Check total duration of profiles
AssertEquals_LREAL(Expected := 0.19429164835544748824, Actual := output.Trajectory.Duration, DELTA := 1E-8, Message := 'Duration incorrect');

// Check duration for each phase
positionExtrema := output.trajectory.profiles[0].positionExtrema();
AssertEquals_LREAL(0.00929214609675180735, positionExtrema.Tmax, 1E-9, message:='Profile[0] Tmax incorrect');
AssertEquals_LREAL(69.55159049131329140891, positionExtrema.Maximum, 1E-9, message:='Profile[0] maximum incorrect');
AssertEquals_LREAL(0.16890359782096156516, positionExtrema.Tmin, 1E-9, message:='Profile[0] Tmin incorrect');
AssertEquals_LREAL(-28.39869225356863324805, positionExtrema.Minimum, 1E-9, message:='Profile[0] minimum incorrect');

positionExtrema := output.trajectory.profiles[1].positionExtrema();
AssertEquals_LREAL(0.00000000000000000000, positionExtrema.Tmax, 1E-9, message:='Profile[1] Tmax incorrect');
AssertEquals_LREAL(-13.39780118806328346182, positionExtrema.Maximum, 1E-9, message:='Profile[1] maximum incorrect');
AssertEquals_LREAL(0.19429164835544748824, positionExtrema.Tmin, 1E-9, message:='Profile[1] Tmin incorrect');
AssertEquals_LREAL(-92.09682308688789476037, positionExtrema.Minimum, 1E-9, message:='Profile[1] minimum incorrect');

positionExtrema := output.trajectory.profiles[2].positionExtrema();
AssertEquals_LREAL(0.15958331587242960414, positionExtrema.Tmax, 1E-9, message:='Profile[2] Tmax incorrect');
AssertEquals_LREAL(-78.59507311744690127853, positionExtrema.Maximum, 1E-9, message:='Profile[2] maximum incorrect');
AssertEquals_LREAL(0.00000000000000000000, positionExtrema.Tmin, 1E-9, message:='Profile[2] Tmin incorrect');
AssertEquals_LREAL(-96.66107573544628905893, positionExtrema.Minimum, 1E-9, message:='Profile[2] minimum incorrect');
   

TEST_FINISHED();
END_METHOD

METHOD Test_Trajectory_62
VAR_INST
  ruckig : Struckig.Ruckig(0.001);
  input : Struckig.InputParameter(3) := (
    Synchronization := SynchronizationType.TimeSync,        
    MaxVelocity := [ 2000.00000000000000000000, 2000.00000000000000000000, 2000.00000000000000000000 ],
    MaxAcceleration := [ 20000.00000000000000000000, 20000.00000000000000000000, 20000.00000000000000000000 ],
    MaxJerk := [ 800000.00000000000000000000, 800000.00000000000000000000, 800000.00000000000000000000 ],
    CurrentPosition := [ 12.59051349490785298713, 2.34116410267218100216, -83.91521339841989401975 ],
    CurrentVelocity := [ -551.49352374949262411974, 694.95621845049936382566, -934.69209805013122149830 ],
    CurrentAcceleration := [ -5149.29503825546817097347, -9527.17655518820902216248, -9641.67382351083688263316 ],
    TargetPosition := [ -69.43235683496359911260, 5.95471336539937112775, -76.71462247839342296629 ],
    TargetVelocity := [ 0.00000000000000000000, 0.00000000000000000000, 0.00000000000000000000 ],
    TargetAcceleration := [ 0.00000000000000000000, 0.00000000000000000000, 0.00000000000000000000 ]
  );
  output : Struckig.OutputParameter;
  positionExtrema : Struckig.PositionExtremaDesc;
END_VAR
TEST('Trajectory_62');

ruckig.update(input, output);

// Check total duration of profiles
AssertEquals_LREAL(Expected := 0.19541920510428964497, Actual := output.Trajectory.Duration, DELTA := 1E-8, Message := 'Duration incorrect');

// Check duration for each phase
positionExtrema := output.trajectory.profiles[0].positionExtrema();
AssertEquals_LREAL(0.00000000000000000000, positionExtrema.Tmax, 1E-9, message:='Profile[0] Tmax incorrect');
AssertEquals_LREAL(12.59051349490785298713, positionExtrema.Maximum, 1E-9, message:='Profile[0] maximum incorrect');
AssertEquals_LREAL(0.19541920510428961721, positionExtrema.Tmin, 1E-9, message:='Profile[0] Tmin incorrect');
AssertEquals_LREAL(-69.43235683496359911260, positionExtrema.Minimum, 1E-9, message:='Profile[0] minimum incorrect');

positionExtrema := output.trajectory.profiles[1].positionExtrema();
AssertEquals_LREAL(0.04065736745126265206, positionExtrema.Tmax, 1E-9, message:='Profile[1] Tmax incorrect');
AssertEquals_LREAL(16.73830873177616496150, positionExtrema.Maximum, 1E-9, message:='Profile[1] maximum incorrect');
AssertEquals_LREAL(0.00000000000000000000, positionExtrema.Tmin, 1E-9, message:='Profile[1] Tmin incorrect');
AssertEquals_LREAL(2.34116410267218100216, positionExtrema.Minimum, 1E-9, message:='Profile[1] minimum incorrect');

positionExtrema := output.trajectory.profiles[2].positionExtrema();
AssertEquals_LREAL(0.19541920510428964497, positionExtrema.Tmax, 1E-9, message:='Profile[2] Tmax incorrect');
AssertEquals_LREAL(-76.71462247839342296629, positionExtrema.Maximum, 1E-9, message:='Profile[2] maximum incorrect');
AssertEquals_LREAL(0.10355548042620135729, positionExtrema.Tmin, 1E-9, message:='Profile[2] Tmin incorrect');
AssertEquals_LREAL(-123.55479709285413036923, positionExtrema.Minimum, 1E-9, message:='Profile[2] minimum incorrect');
   

TEST_FINISHED();
END_METHOD

METHOD Test_Trajectory_HasTargetAcceleration_63
VAR_INST
  ruckig : Struckig.Ruckig(0.001);
  input : Struckig.InputParameter(3) := (
    Synchronization := SynchronizationType.TimeSync,        
    MaxVelocity := [ 2000.00000000000000000000, 2000.00000000000000000000, 2000.00000000000000000000 ],
    MaxAcceleration := [ 20000.00000000000000000000, 20000.00000000000000000000, 20000.00000000000000000000 ],
    MaxJerk := [ 800000.00000000000000000000, 800000.00000000000000000000, 800000.00000000000000000000 ],
    CurrentPosition := [ 92.10487433807648471884, 89.01461536061293600142, 43.32328991111594973518 ],
    CurrentVelocity := [ 582.24588381700414174702, -343.03367241945181831397, -453.35877163487862162583 ],
    CurrentAcceleration := [ -2628.64665337560109037440, 4464.34448190908915421460, 7008.64234603228396736085 ],
    TargetPosition := [ 92.91310177759680755116, 56.54940187438580778689, 5.30614662549113802470 ],
    TargetVelocity := [ 0.00000000000000000000, 0.00000000000000000000, 0.00000000000000000000 ],
    TargetAcceleration := [ -858.57813559612441167701, 114.62677054353116545826, 120.82597031040290858073 ]
  );
  output : Struckig.OutputParameter;
  positionExtrema : Struckig.PositionExtremaDesc;
END_VAR
TEST('Trajectory_HasTargetAcceleration_63');

ruckig.update(input, output);

// Check total duration of profiles
AssertEquals_LREAL(Expected := 0.10861795461857774725, Actual := output.Trajectory.Duration, DELTA := 1E-8, Message := 'Duration incorrect');

